(* Logix 5000 project; controller reports 1756-L63 rev 20.15; software revision 20.04; part 13 of 52 *)

        [466].log_data[0].valid := 1, [466].log_data[1].valid := 1, [466].log_data[2].valid := 1, [466].log_data[3].valid := 1, [466].log_data[4].valid := 1, [466].log_data[5].valid := 1, [466].log_data[6].valid := 1, [466].log_data[7].valid := 1, [466].log_data[8].valid := 1, [466].log_data[9].valid := 1, [466].log_data[10].valid := 1, [466].log_data[11].valid := 1, [466].log_data[12].valid := 1, [466].log_data[13].valid := 1, [466].log_data[14].valid := 1, [466].log_data[15].valid := 1, [466].log_data[16].valid := 1, [466].log_data[17].valid := 1, [466].log_data[18].valid := 1, [466].log_data[19].valid := 1, [466].time.Year := 2023, [466].time.Month := 1, [466].time.Day := 19, [466].time.Hour := 15, [466].time.Minute := 14, [466].time.Second := 59, [467].log_data[0].min := 1.0, [467].log_data[0].max := 1.0, [467].log_data[0].total := 300.0, [467].log_data[0].time := 300.0, [467].log_data[0].minminute := 15, [467].log_data[0].maxminute := 15, [467].log_data[0].valid := 1, [467].log_data[1].valid := 1, [467].log_data[2].valid := 1, [467].log_data[3].valid := 1, [467].log_data[4].valid := 1, [467].log_data[5].valid := 1, [467].log_data[6].valid := 1, [467].log_data[7].valid := 1, [467].log_data[8].valid := 1, [467].log_data[9].valid := 1, [467].log_data[10].valid := 1, [467].log_data[11].valid := 1, [467].log_data[12].valid := 1, [467].log_data[13].valid := 1, [467].log_data[14].valid := 1, [467].log_data[15].valid := 1, [467].log_data[16].valid := 1, [467].log_data[17].valid := 1, [467].log_data[18].valid := 1, [467].log_data[19].valid := 1, [467].time.Year := 2023, [467].time.Month := 1, [467].time.Day := 19, [467].time.Hour := 15, [467].time.Minute := 19, [467].time.Second := 59, [468].log_data[0].min := 1.0, [468].log_data[0].max := 1.0,
        [468].log_data[0].total := 300.0, [468].log_data[0].time := 300.0, [468].log_data[0].minminute := 20, [468].log_data[0].maxminute := 20, [468].log_data[0].valid := 1, [468].log_data[1].valid := 1, [468].log_data[2].valid := 1, [468].log_data[3].valid := 1, [468].log_data[4].valid := 1, [468].log_data[5].valid := 1, [468].log_data[6].valid := 1, [468].log_data[7].valid := 1, [468].log_data[8].valid := 1, [468].log_data[9].valid := 1, [468].log_data[10].valid := 1, [468].log_data[11].valid := 1, [468].log_data[12].valid := 1, [468].log_data[13].valid := 1, [468].log_data[14].valid := 1, [468].log_data[15].valid := 1, [468].log_data[16].valid := 1, [468].log_data[17].valid := 1, [468].log_data[18].valid := 1, [468].log_data[19].valid := 1, [468].time.Year := 2023, [468].time.Month := 1, [468].time.Day := 19, [468].time.Hour := 15, [468].time.Minute := 24, [468].time.Second := 59, [469].log_data[0].min := 1.0, [469].log_data[0].max := 1.0, [469].log_data[0].total := 44.5, [469].log_data[0].time := 44.5, [469].log_data[0].minminute := 25, [469].log_data[0].maxminute := 25, [469].log_data[0].valid := 1, [469].log_data[1].valid := 1, [469].log_data[2].valid := 1, [469].log_data[3].valid := 1, [469].log_data[4].valid := 1, [469].log_data[5].valid := 1, [469].log_data[6].valid := 1, [469].log_data[7].valid := 1, [469].log_data[8].valid := 1, [469].log_data[9].valid := 1, [469].log_data[10].valid := 1, [469].log_data[11].valid := 1, [469].log_data[12].valid := 1, [469].log_data[13].valid := 1, [469].log_data[14].valid := 1, [469].log_data[15].valid := 1, [469].log_data[16].valid := 1, [469].log_data[17].valid := 1, [469].log_data[18].valid := 1, [469].log_data[19].valid := 1, [470].log_data[0].min := 1.0, [470].log_data[0].max := 1.0, [470].log_data[0].total := 300.0, [470].log_data[0].time := 300.0,
        [470].log_data[0].minminute := 30, [470].log_data[0].maxminute := 30, [470].log_data[0].valid := 1, [470].log_data[1].valid := 1, [470].log_data[2].valid := 1, [470].log_data[3].valid := 1, [470].log_data[4].valid := 1, [470].log_data[5].valid := 1, [470].log_data[6].valid := 1, [470].log_data[7].valid := 1, [470].log_data[8].valid := 1, [470].log_data[9].valid := 1, [470].log_data[10].valid := 1, [470].log_data[11].valid := 1, [470].log_data[12].valid := 1, [470].log_data[13].valid := 1, [470].log_data[14].valid := 1, [470].log_data[15].valid := 1, [470].log_data[16].valid := 1, [470].log_data[17].valid := 1, [470].log_data[18].valid := 1, [470].log_data[19].valid := 1, [470].time.Year := 2023, [470].time.Month := 1, [470].time.Day := 11, [470].time.Hour := 7, [470].time.Minute := 34, [470].time.Second := 59, [471].log_data[0].min := 1.0, [471].log_data[0].max := 1.0, [471].log_data[0].total := 300.0, [471].log_data[0].time := 300.0, [471].log_data[0].minminute := 35, [471].log_data[0].maxminute := 35, [471].log_data[0].valid := 1, [471].log_data[1].valid := 1, [471].log_data[2].valid := 1, [471].log_data[3].valid := 1, [471].log_data[4].valid := 1, [471].log_data[5].valid := 1, [471].log_data[6].valid := 1, [471].log_data[7].valid := 1, [471].log_data[8].valid := 1, [471].log_data[9].valid := 1, [471].log_data[10].valid := 1, [471].log_data[11].valid := 1, [471].log_data[12].valid := 1, [471].log_data[13].valid := 1, [471].log_data[14].valid := 1, [471].log_data[15].valid := 1, [471].log_data[16].valid := 1, [471].log_data[17].valid := 1, [471].log_data[18].valid := 1, [471].log_data[19].valid := 1, [471].time.Year := 2023, [471].time.Month := 1, [471].time.Day := 11, [471].time.Hour := 7, [471].time.Minute := 39, [471].time.Second := 59,
        [472].log_data[0].min := 1.0, [472].log_data[0].max := 1.0, [472].log_data[0].total := 300.0, [472].log_data[0].time := 300.0, [472].log_data[0].minminute := 40, [472].log_data[0].maxminute := 40, [472].log_data[0].valid := 1, [472].log_data[1].valid := 1, [472].log_data[2].valid := 1, [472].log_data[3].valid := 1, [472].log_data[4].valid := 1, [472].log_data[5].valid := 1, [472].log_data[6].valid := 1, [472].log_data[7].valid := 1, [472].log_data[8].valid := 1, [472].log_data[9].valid := 1, [472].log_data[10].valid := 1, [472].log_data[11].valid := 1, [472].log_data[12].valid := 1, [472].log_data[13].valid := 1, [472].log_data[14].valid := 1, [472].log_data[15].valid := 1, [472].log_data[16].valid := 1, [472].log_data[17].valid := 1, [472].log_data[18].valid := 1, [472].log_data[19].valid := 1, [472].time.Year := 2023, [472].time.Month := 1, [472].time.Day := 11, [472].time.Hour := 7, [472].time.Minute := 44, [472].time.Second := 59, [473].log_data[0].min := 1.0, [473].log_data[0].max := 1.0, [473].log_data[0].total := 300.0, [473].log_data[0].time := 300.0, [473].log_data[0].minminute := 45, [473].log_data[0].maxminute := 45, [473].log_data[0].valid := 1, [473].log_data[1].valid := 1, [473].log_data[2].valid := 1, [473].log_data[3].valid := 1, [473].log_data[4].valid := 1, [473].log_data[5].valid := 1, [473].log_data[6].valid := 1, [473].log_data[7].valid := 1, [473].log_data[8].valid := 1, [473].log_data[9].valid := 1, [473].log_data[10].valid := 1, [473].log_data[11].valid := 1, [473].log_data[12].valid := 1, [473].log_data[13].valid := 1, [473].log_data[14].valid := 1, [473].log_data[15].valid := 1, [473].log_data[16].valid := 1, [473].log_data[17].valid := 1, [473].log_data[18].valid := 1, [473].log_data[19].valid := 1, [473].time.Year := 2023, [473].time.Month := 1,
        [473].time.Day := 11, [473].time.Hour := 7, [473].time.Minute := 49, [473].time.Second := 59, [474].log_data[0].min := 1.0, [474].log_data[0].max := 1.0, [474].log_data[0].total := 300.0, [474].log_data[0].time := 300.0, [474].log_data[0].minminute := 50, [474].log_data[0].maxminute := 50, [474].log_data[0].valid := 1, [474].log_data[1].valid := 1, [474].log_data[2].valid := 1, [474].log_data[3].valid := 1, [474].log_data[4].valid := 1, [474].log_data[5].valid := 1, [474].log_data[6].valid := 1, [474].log_data[7].valid := 1, [474].log_data[8].valid := 1, [474].log_data[9].valid := 1, [474].log_data[10].valid := 1, [474].log_data[11].valid := 1, [474].log_data[12].valid := 1, [474].log_data[13].valid := 1, [474].log_data[14].valid := 1, [474].log_data[15].valid := 1, [474].log_data[16].valid := 1, [474].log_data[17].valid := 1, [474].log_data[18].valid := 1, [474].log_data[19].valid := 1, [474].time.Year := 2023, [474].time.Month := 1, [474].time.Day := 11, [474].time.Hour := 7, [474].time.Minute := 54, [474].time.Second := 59, [475].log_data[0].min := 1.0, [475].log_data[0].max := 1.0, [475].log_data[0].total := 300.0, [475].log_data[0].time := 300.0, [475].log_data[0].minminute := 55, [475].log_data[0].maxminute := 55, [475].log_data[0].valid := 1, [475].log_data[1].valid := 1, [475].log_data[2].valid := 1, [475].log_data[3].valid := 1, [475].log_data[4].valid := 1, [475].log_data[5].valid := 1, [475].log_data[6].valid := 1, [475].log_data[7].valid := 1, [475].log_data[8].valid := 1, [475].log_data[9].valid := 1, [475].log_data[10].valid := 1, [475].log_data[11].valid := 1, [475].log_data[12].valid := 1, [475].log_data[13].valid := 1, [475].log_data[14].valid := 1, [475].log_data[15].valid := 1, [475].log_data[16].valid := 1, [475].log_data[17].valid := 1,
        [475].log_data[18].valid := 1, [475].log_data[19].valid := 1, [475].time.Year := 2023, [475].time.Month := 1, [475].time.Day := 11, [475].time.Hour := 7, [475].time.Minute := 59, [475].time.Second := 59, [476].log_data[0].min := 1.0, [476].log_data[0].max := 1.0, [476].log_data[0].total := 300.0, [476].log_data[0].time := 300.0, [476].log_data[0].valid := 1, [476].log_data[1].valid := 1, [476].log_data[2].valid := 1, [476].log_data[3].valid := 1, [476].log_data[4].valid := 1, [476].log_data[5].valid := 1, [476].log_data[6].valid := 1, [476].log_data[7].valid := 1, [476].log_data[8].valid := 1, [476].log_data[9].valid := 1, [476].log_data[10].valid := 1, [476].log_data[11].valid := 1, [476].log_data[12].valid := 1, [476].log_data[13].valid := 1, [476].log_data[14].valid := 1, [476].log_data[15].valid := 1, [476].log_data[16].valid := 1, [476].log_data[17].valid := 1, [476].log_data[18].valid := 1, [476].log_data[19].valid := 1, [476].time.Year := 2023, [476].time.Month := 1, [476].time.Day := 11, [476].time.Hour := 8, [476].time.Minute := 4, [476].time.Second := 59, [477].log_data[0].min := 1.0, [477].log_data[0].max := 1.0, [477].log_data[0].total := 300.0, [477].log_data[0].time := 300.0, [477].log_data[0].minminute := 5, [477].log_data[0].maxminute := 5, [477].log_data[0].valid := 1, [477].log_data[1].valid := 1, [477].log_data[2].valid := 1, [477].log_data[3].valid := 1, [477].log_data[4].valid := 1, [477].log_data[5].valid := 1, [477].log_data[6].valid := 1, [477].log_data[7].valid := 1, [477].log_data[8].valid := 1, [477].log_data[9].valid := 1, [477].log_data[10].valid := 1, [477].log_data[11].valid := 1, [477].log_data[12].valid := 1, [477].log_data[13].valid := 1, [477].log_data[14].valid := 1, [477].log_data[15].valid := 1,
        [477].log_data[16].valid := 1, [477].log_data[17].valid := 1, [477].log_data[18].valid := 1, [477].log_data[19].valid := 1, [477].time.Year := 2023, [477].time.Month := 1, [477].time.Day := 11, [477].time.Hour := 8, [477].time.Minute := 9, [477].time.Second := 59, [478].log_data[0].min := 1.0, [478].log_data[0].max := 1.0, [478].log_data[0].total := 300.0, [478].log_data[0].time := 300.0, [478].log_data[0].minminute := 10, [478].log_data[0].maxminute := 10, [478].log_data[0].valid := 1, [478].log_data[1].valid := 1, [478].log_data[2].valid := 1, [478].log_data[3].valid := 1, [478].log_data[4].valid := 1, [478].log_data[5].valid := 1, [478].log_data[6].valid := 1, [478].log_data[7].valid := 1, [478].log_data[8].valid := 1, [478].log_data[9].valid := 1, [478].log_data[10].valid := 1, [478].log_data[11].valid := 1, [478].log_data[12].valid := 1, [478].log_data[13].valid := 1, [478].log_data[14].valid := 1, [478].log_data[15].valid := 1, [478].log_data[16].valid := 1, [478].log_data[17].valid := 1, [478].log_data[18].valid := 1, [478].log_data[19].valid := 1, [478].time.Year := 2023, [478].time.Month := 1, [478].time.Day := 11, [478].time.Hour := 8, [478].time.Minute := 14, [478].time.Second := 59, [479].log_data[0].min := 1.0, [479].log_data[0].max := 1.0, [479].log_data[0].total := 300.0, [479].log_data[0].time := 300.0, [479].log_data[0].minminute := 15, [479].log_data[0].maxminute := 15, [479].log_data[0].valid := 1, [479].log_data[1].valid := 1, [479].log_data[2].valid := 1, [479].log_data[3].valid := 1, [479].log_data[4].valid := 1, [479].log_data[5].valid := 1, [479].log_data[6].valid := 1, [479].log_data[7].valid := 1, [479].log_data[8].valid := 1, [479].log_data[9].valid := 1, [479].log_data[10].valid := 1, [479].log_data[11].valid := 1,
        [479].log_data[12].valid := 1, [479].log_data[13].valid := 1, [479].log_data[14].valid := 1, [479].log_data[15].valid := 1, [479].log_data[16].valid := 1, [479].log_data[17].valid := 1, [479].log_data[18].valid := 1, [479].log_data[19].valid := 1, [479].time.Year := 2023, [479].time.Month := 1, [479].time.Day := 11, [479].time.Hour := 8, [479].time.Minute := 19, [479].time.Second := 59, [480].log_data[0].min := 1.0, [480].log_data[0].max := 1.0, [480].log_data[0].total := 300.0, [480].log_data[0].time := 300.0, [480].log_data[0].minminute := 20, [480].log_data[0].maxminute := 20, [480].log_data[0].valid := 1, [480].log_data[1].valid := 1, [480].log_data[2].valid := 1, [480].log_data[3].valid := 1, [480].log_data[4].valid := 1, [480].log_data[5].valid := 1, [480].log_data[6].valid := 1, [480].log_data[7].valid := 1, [480].log_data[8].valid := 1, [480].log_data[9].valid := 1, [480].log_data[10].valid := 1, [480].log_data[11].valid := 1, [480].log_data[12].valid := 1, [480].log_data[13].valid := 1, [480].log_data[14].valid := 1, [480].log_data[15].valid := 1, [480].log_data[16].valid := 1, [480].log_data[17].valid := 1, [480].log_data[18].valid := 1, [480].log_data[19].valid := 1, [480].time.Year := 2023, [480].time.Month := 1, [480].time.Day := 11, [480].time.Hour := 8, [480].time.Minute := 24, [480].time.Second := 59, [481].log_data[0].min := 1.0, [481].log_data[0].max := 1.0, [481].log_data[0].total := 300.0, [481].log_data[0].time := 300.0, [481].log_data[0].minminute := 25, [481].log_data[0].maxminute := 25, [481].log_data[0].valid := 1, [481].log_data[1].valid := 1, [481].log_data[2].valid := 1, [481].log_data[3].valid := 1, [481].log_data[4].valid := 1, [481].log_data[5].valid := 1, [481].log_data[6].valid := 1, [481].log_data[7].valid := 1,
        [481].log_data[8].valid := 1, [481].log_data[9].valid := 1, [481].log_data[10].valid := 1, [481].log_data[11].valid := 1, [481].log_data[12].valid := 1, [481].log_data[13].valid := 1, [481].log_data[14].valid := 1, [481].log_data[15].valid := 1, [481].log_data[16].valid := 1, [481].log_data[17].valid := 1, [481].log_data[18].valid := 1, [481].log_data[19].valid := 1, [481].time.Year := 2023, [481].time.Month := 1, [481].time.Day := 11, [481].time.Hour := 8, [481].time.Minute := 29, [481].time.Second := 59, [482].log_data[0].min := 1.0, [482].log_data[0].max := 1.0, [482].log_data[0].total := 300.0, [482].log_data[0].time := 300.0, [482].log_data[0].minminute := 30, [482].log_data[0].maxminute := 30, [482].log_data[0].valid := 1, [482].log_data[1].valid := 1, [482].log_data[2].valid := 1, [482].log_data[3].valid := 1, [482].log_data[4].valid := 1, [482].log_data[5].valid := 1, [482].log_data[6].valid := 1, [482].log_data[7].valid := 1, [482].log_data[8].valid := 1, [482].log_data[9].valid := 1, [482].log_data[10].valid := 1, [482].log_data[11].valid := 1, [482].log_data[12].valid := 1, [482].log_data[13].valid := 1, [482].log_data[14].valid := 1, [482].log_data[15].valid := 1, [482].log_data[16].valid := 1, [482].log_data[17].valid := 1, [482].log_data[18].valid := 1, [482].log_data[19].valid := 1, [482].time.Year := 2023, [482].time.Month := 1, [482].time.Day := 11, [482].time.Hour := 8, [482].time.Minute := 34, [482].time.Second := 59, [483].log_data[0].min := 1.0, [483].log_data[0].max := 1.0, [483].log_data[0].total := 300.0, [483].log_data[0].time := 300.0, [483].log_data[0].minminute := 35, [483].log_data[0].maxminute := 35, [483].log_data[0].valid := 1, [483].log_data[1].valid := 1, [483].log_data[2].valid := 1, [483].log_data[3].valid := 1,
        [483].log_data[4].valid := 1, [483].log_data[5].valid := 1, [483].log_data[6].valid := 1, [483].log_data[7].valid := 1, [483].log_data[8].valid := 1, [483].log_data[9].valid := 1, [483].log_data[10].valid := 1, [483].log_data[11].valid := 1, [483].log_data[12].valid := 1, [483].log_data[13].valid := 1, [483].log_data[14].valid := 1, [483].log_data[15].valid := 1, [483].log_data[16].valid := 1, [483].log_data[17].valid := 1, [483].log_data[18].valid := 1, [483].log_data[19].valid := 1, [483].time.Year := 2023, [483].time.Month := 1, [483].time.Day := 11, [483].time.Hour := 8, [483].time.Minute := 39, [483].time.Second := 59, [484].log_data[0].min := 1.0, [484].log_data[0].max := 1.0, [484].log_data[0].total := 300.0, [484].log_data[0].time := 300.0, [484].log_data[0].minminute := 40, [484].log_data[0].maxminute := 40, [484].log_data[0].valid := 1, [484].log_data[1].valid := 1, [484].log_data[2].valid := 1, [484].log_data[3].valid := 1, [484].log_data[4].valid := 1, [484].log_data[5].valid := 1, [484].log_data[6].valid := 1, [484].log_data[7].valid := 1, [484].log_data[8].valid := 1, [484].log_data[9].valid := 1, [484].log_data[10].valid := 1, [484].log_data[11].valid := 1, [484].log_data[12].valid := 1, [484].log_data[13].valid := 1, [484].log_data[14].valid := 1, [484].log_data[15].valid := 1, [484].log_data[16].valid := 1, [484].log_data[17].valid := 1, [484].log_data[18].valid := 1, [484].log_data[19].valid := 1, [484].time.Year := 2023, [484].time.Month := 1, [484].time.Day := 11, [484].time.Hour := 8, [484].time.Minute := 44, [484].time.Second := 59, [485].log_data[0].min := 1.0, [485].log_data[0].max := 1.0, [485].log_data[0].total := 300.0, [485].log_data[0].time := 300.0, [485].log_data[0].minminute := 45, [485].log_data[0].maxminute := 45,
        [485].log_data[0].valid := 1, [485].log_data[1].valid := 1, [485].log_data[2].valid := 1, [485].log_data[3].valid := 1, [485].log_data[4].valid := 1, [485].log_data[5].valid := 1, [485].log_data[6].valid := 1, [485].log_data[7].valid := 1, [485].log_data[8].valid := 1, [485].log_data[9].valid := 1, [485].log_data[10].valid := 1, [485].log_data[11].valid := 1, [485].log_data[12].valid := 1, [485].log_data[13].valid := 1, [485].log_data[14].valid := 1, [485].log_data[15].valid := 1, [485].log_data[16].valid := 1, [485].log_data[17].valid := 1, [485].log_data[18].valid := 1, [485].log_data[19].valid := 1, [485].time.Year := 2023, [485].time.Month := 1, [485].time.Day := 11, [485].time.Hour := 8, [485].time.Minute := 49, [485].time.Second := 59, [486].log_data[0].min := 1.0, [486].log_data[0].max := 1.0, [486].log_data[0].total := 300.0, [486].log_data[0].time := 300.0, [486].log_data[0].minminute := 50, [486].log_data[0].maxminute := 50, [486].log_data[0].valid := 1, [486].log_data[1].valid := 1, [486].log_data[2].valid := 1, [486].log_data[3].valid := 1, [486].log_data[4].valid := 1, [486].log_data[5].valid := 1, [486].log_data[6].valid := 1, [486].log_data[7].valid := 1, [486].log_data[8].valid := 1, [486].log_data[9].valid := 1, [486].log_data[10].valid := 1, [486].log_data[11].valid := 1, [486].log_data[12].valid := 1, [486].log_data[13].valid := 1, [486].log_data[14].valid := 1, [486].log_data[15].valid := 1, [486].log_data[16].valid := 1, [486].log_data[17].valid := 1, [486].log_data[18].valid := 1, [486].log_data[19].valid := 1, [486].time.Year := 2023, [486].time.Month := 1, [486].time.Day := 11, [486].time.Hour := 8, [486].time.Minute := 54, [486].time.Second := 59, [487].log_data[0].min := 1.0, [487].log_data[0].max := 1.0,
        [487].log_data[0].total := 300.0, [487].log_data[0].time := 300.0, [487].log_data[0].minminute := 55, [487].log_data[0].maxminute := 55, [487].log_data[0].valid := 1, [487].log_data[1].valid := 1, [487].log_data[2].valid := 1, [487].log_data[3].valid := 1, [487].log_data[4].valid := 1, [487].log_data[5].valid := 1, [487].log_data[6].valid := 1, [487].log_data[7].valid := 1, [487].log_data[8].valid := 1, [487].log_data[9].valid := 1, [487].log_data[10].valid := 1, [487].log_data[11].valid := 1, [487].log_data[12].valid := 1, [487].log_data[13].valid := 1, [487].log_data[14].valid := 1, [487].log_data[15].valid := 1, [487].log_data[16].valid := 1, [487].log_data[17].valid := 1, [487].log_data[18].valid := 1, [487].log_data[19].valid := 1, [487].time.Year := 2023, [487].time.Month := 1, [487].time.Day := 11, [487].time.Hour := 8, [487].time.Minute := 59, [487].time.Second := 59, [488].log_data[0].min := 1.0, [488].log_data[0].max := 1.0, [488].log_data[0].total := 300.0, [488].log_data[0].time := 300.0, [488].log_data[0].valid := 1, [488].log_data[1].valid := 1, [488].log_data[2].valid := 1, [488].log_data[3].valid := 1, [488].log_data[4].valid := 1, [488].log_data[5].valid := 1, [488].log_data[6].valid := 1, [488].log_data[7].valid := 1, [488].log_data[8].valid := 1, [488].log_data[9].valid := 1, [488].log_data[10].valid := 1, [488].log_data[11].valid := 1, [488].log_data[12].valid := 1, [488].log_data[13].valid := 1, [488].log_data[14].valid := 1, [488].log_data[15].valid := 1, [488].log_data[16].valid := 1, [488].log_data[17].valid := 1, [488].log_data[18].valid := 1, [488].log_data[19].valid := 1, [488].time.Year := 2023, [488].time.Month := 1, [488].time.Day := 11, [488].time.Hour := 9, [488].time.Minute := 4, [488].time.Second := 59,
        [489].log_data[0].min := 1.0, [489].log_data[0].max := 1.0, [489].log_data[0].total := 300.0, [489].log_data[0].time := 300.0, [489].log_data[0].minminute := 5, [489].log_data[0].maxminute := 5, [489].log_data[0].valid := 1, [489].log_data[1].valid := 1, [489].log_data[2].valid := 1, [489].log_data[3].valid := 1, [489].log_data[4].valid := 1, [489].log_data[5].valid := 1, [489].log_data[6].valid := 1, [489].log_data[7].valid := 1, [489].log_data[8].valid := 1, [489].log_data[9].valid := 1, [489].log_data[10].valid := 1, [489].log_data[11].valid := 1, [489].log_data[12].valid := 1, [489].log_data[13].valid := 1, [489].log_data[14].valid := 1, [489].log_data[15].valid := 1, [489].log_data[16].valid := 1, [489].log_data[17].valid := 1, [489].log_data[18].valid := 1, [489].log_data[19].valid := 1, [489].time.Year := 2023, [489].time.Month := 1, [489].time.Day := 11, [489].time.Hour := 9, [489].time.Minute := 9, [489].time.Second := 59, [490].log_data[0].min := 1.0, [490].log_data[0].max := 1.0, [490].log_data[0].total := 300.0, [490].log_data[0].time := 300.0, [490].log_data[0].minminute := 10, [490].log_data[0].maxminute := 10, [490].log_data[0].valid := 1, [490].log_data[1].valid := 1, [490].log_data[2].valid := 1, [490].log_data[3].valid := 1, [490].log_data[4].valid := 1, [490].log_data[5].valid := 1, [490].log_data[6].valid := 1, [490].log_data[7].valid := 1, [490].log_data[8].valid := 1, [490].log_data[9].valid := 1, [490].log_data[10].valid := 1, [490].log_data[11].valid := 1, [490].log_data[12].valid := 1, [490].log_data[13].valid := 1, [490].log_data[14].valid := 1, [490].log_data[15].valid := 1, [490].log_data[16].valid := 1, [490].log_data[17].valid := 1, [490].log_data[18].valid := 1, [490].log_data[19].valid := 1, [490].time.Year := 2023, [490].time.Month := 1,
        [490].time.Day := 11, [490].time.Hour := 9, [490].time.Minute := 14, [490].time.Second := 59, [491].log_data[0].min := 1.0, [491].log_data[0].max := 1.0, [491].log_data[0].total := 300.0, [491].log_data[0].time := 300.0, [491].log_data[0].minminute := 15, [491].log_data[0].maxminute := 15, [491].log_data[0].valid := 1, [491].log_data[1].valid := 1, [491].log_data[2].valid := 1, [491].log_data[3].valid := 1, [491].log_data[4].valid := 1, [491].log_data[5].valid := 1, [491].log_data[6].valid := 1, [491].log_data[7].valid := 1, [491].log_data[8].valid := 1, [491].log_data[9].valid := 1, [491].log_data[10].valid := 1, [491].log_data[11].valid := 1, [491].log_data[12].valid := 1, [491].log_data[13].valid := 1, [491].log_data[14].valid := 1, [491].log_data[15].valid := 1, [491].log_data[16].valid := 1, [491].log_data[17].valid := 1, [491].log_data[18].valid := 1, [491].log_data[19].valid := 1, [491].time.Year := 2023, [491].time.Month := 1, [491].time.Day := 11, [491].time.Hour := 9, [491].time.Minute := 19, [491].time.Second := 59, [492].log_data[0].min := 1.0, [492].log_data[0].max := 1.0, [492].log_data[0].total := 300.0, [492].log_data[0].time := 300.0, [492].log_data[0].minminute := 20, [492].log_data[0].maxminute := 20, [492].log_data[0].valid := 1, [492].log_data[1].valid := 1, [492].log_data[2].valid := 1, [492].log_data[3].valid := 1, [492].log_data[4].valid := 1, [492].log_data[5].valid := 1, [492].log_data[6].valid := 1, [492].log_data[7].valid := 1, [492].log_data[8].valid := 1, [492].log_data[9].valid := 1, [492].log_data[10].valid := 1, [492].log_data[11].valid := 1, [492].log_data[12].valid := 1, [492].log_data[13].valid := 1, [492].log_data[14].valid := 1, [492].log_data[15].valid := 1, [492].log_data[16].valid := 1, [492].log_data[17].valid := 1,
        [492].log_data[18].valid := 1, [492].log_data[19].valid := 1, [492].time.Year := 2023, [492].time.Month := 1, [492].time.Day := 11, [492].time.Hour := 9, [492].time.Minute := 24, [492].time.Second := 59, [493].log_data[0].min := 1.0, [493].log_data[0].max := 1.0, [493].log_data[0].total := 300.0, [493].log_data[0].time := 300.0, [493].log_data[0].minminute := 25, [493].log_data[0].maxminute := 25, [493].log_data[0].valid := 1, [493].log_data[1].valid := 1, [493].log_data[2].valid := 1, [493].log_data[3].valid := 1, [493].log_data[4].valid := 1, [493].log_data[5].valid := 1, [493].log_data[6].valid := 1, [493].log_data[7].valid := 1, [493].log_data[8].valid := 1, [493].log_data[9].valid := 1, [493].log_data[10].valid := 1, [493].log_data[11].valid := 1, [493].log_data[12].valid := 1, [493].log_data[13].valid := 1, [493].log_data[14].valid := 1, [493].log_data[15].valid := 1, [493].log_data[16].valid := 1, [493].log_data[17].valid := 1, [493].log_data[18].valid := 1, [493].log_data[19].valid := 1, [493].time.Year := 2023, [493].time.Month := 1, [493].time.Day := 11, [493].time.Hour := 9, [493].time.Minute := 29, [493].time.Second := 59, [494].log_data[0].min := 1.0, [494].log_data[0].max := 1.0, [494].log_data[0].total := 300.0, [494].log_data[0].time := 300.0, [494].log_data[0].minminute := 30, [494].log_data[0].maxminute := 30, [494].log_data[0].valid := 1, [494].log_data[1].valid := 1, [494].log_data[2].valid := 1, [494].log_data[3].valid := 1, [494].log_data[4].valid := 1, [494].log_data[5].valid := 1, [494].log_data[6].valid := 1, [494].log_data[7].valid := 1, [494].log_data[8].valid := 1, [494].log_data[9].valid := 1, [494].log_data[10].valid := 1, [494].log_data[11].valid := 1, [494].log_data[12].valid := 1, [494].log_data[13].valid := 1,
        [494].log_data[14].valid := 1, [494].log_data[15].valid := 1, [494].log_data[16].valid := 1, [494].log_data[17].valid := 1, [494].log_data[18].valid := 1, [494].log_data[19].valid := 1, [494].time.Year := 2023, [494].time.Month := 1, [494].time.Day := 11, [494].time.Hour := 9, [494].time.Minute := 34, [494].time.Second := 59, [495].log_data[0].min := 1.0, [495].log_data[0].max := 1.0, [495].log_data[0].total := 300.0, [495].log_data[0].time := 300.0, [495].log_data[0].minminute := 35, [495].log_data[0].maxminute := 35, [495].log_data[0].valid := 1, [495].log_data[1].valid := 1, [495].log_data[2].valid := 1, [495].log_data[3].valid := 1, [495].log_data[4].valid := 1, [495].log_data[5].valid := 1, [495].log_data[6].valid := 1, [495].log_data[7].valid := 1, [495].log_data[8].valid := 1, [495].log_data[9].valid := 1, [495].log_data[10].valid := 1, [495].log_data[11].valid := 1, [495].log_data[12].valid := 1, [495].log_data[13].valid := 1, [495].log_data[14].valid := 1, [495].log_data[15].valid := 1, [495].log_data[16].valid := 1, [495].log_data[17].valid := 1, [495].log_data[18].valid := 1, [495].log_data[19].valid := 1, [495].time.Year := 2023, [495].time.Month := 1, [495].time.Day := 11, [495].time.Hour := 9, [495].time.Minute := 39, [495].time.Second := 59, [496].log_data[0].min := 1.0, [496].log_data[0].max := 1.0, [496].log_data[0].total := 300.0, [496].log_data[0].time := 300.0, [496].log_data[0].minminute := 40, [496].log_data[0].maxminute := 40, [496].log_data[0].valid := 1, [496].log_data[1].valid := 1, [496].log_data[2].valid := 1, [496].log_data[3].valid := 1, [496].log_data[4].valid := 1, [496].log_data[5].valid := 1, [496].log_data[6].valid := 1, [496].log_data[7].valid := 1, [496].log_data[8].valid := 1, [496].log_data[9].valid := 1,
        [496].log_data[10].valid := 1, [496].log_data[11].valid := 1, [496].log_data[12].valid := 1, [496].log_data[13].valid := 1, [496].log_data[14].valid := 1, [496].log_data[15].valid := 1, [496].log_data[16].valid := 1, [496].log_data[17].valid := 1, [496].log_data[18].valid := 1, [496].log_data[19].valid := 1, [496].time.Year := 2023, [496].time.Month := 1, [496].time.Day := 11, [496].time.Hour := 9, [496].time.Minute := 44, [496].time.Second := 59, [497].log_data[0].min := 1.0, [497].log_data[0].max := 1.0, [497].log_data[0].total := 300.0, [497].log_data[0].time := 300.0, [497].log_data[0].minminute := 45, [497].log_data[0].maxminute := 45, [497].log_data[0].valid := 1, [497].log_data[1].valid := 1, [497].log_data[2].valid := 1, [497].log_data[3].valid := 1, [497].log_data[4].valid := 1, [497].log_data[5].valid := 1, [497].log_data[6].valid := 1, [497].log_data[7].valid := 1, [497].log_data[8].valid := 1, [497].log_data[9].valid := 1, [497].log_data[10].valid := 1, [497].log_data[11].valid := 1, [497].log_data[12].valid := 1, [497].log_data[13].valid := 1, [497].log_data[14].valid := 1, [497].log_data[15].valid := 1, [497].log_data[16].valid := 1, [497].log_data[17].valid := 1, [497].log_data[18].valid := 1, [497].log_data[19].valid := 1, [497].time.Year := 2023, [497].time.Month := 1, [497].time.Day := 11, [497].time.Hour := 9, [497].time.Minute := 49, [497].time.Second := 59, [498].log_data[0].min := 1.0, [498].log_data[0].max := 1.0, [498].log_data[0].total := 300.0, [498].log_data[0].time := 300.0, [498].log_data[0].minminute := 50, [498].log_data[0].maxminute := 50, [498].log_data[0].valid := 1, [498].log_data[1].valid := 1, [498].log_data[2].valid := 1, [498].log_data[3].valid := 1, [498].log_data[4].valid := 1, [498].log_data[5].valid := 1,
        [498].log_data[6].valid := 1, [498].log_data[7].valid := 1, [498].log_data[8].valid := 1, [498].log_data[9].valid := 1, [498].log_data[10].valid := 1, [498].log_data[11].valid := 1, [498].log_data[12].valid := 1, [498].log_data[13].valid := 1, [498].log_data[14].valid := 1, [498].log_data[15].valid := 1, [498].log_data[16].valid := 1, [498].log_data[17].valid := 1, [498].log_data[18].valid := 1, [498].log_data[19].valid := 1, [498].time.Year := 2023, [498].time.Month := 1, [498].time.Day := 11, [498].time.Hour := 9, [498].time.Minute := 54, [498].time.Second := 59, [499].log_data[0].min := 1.0, [499].log_data[0].max := 1.0, [499].log_data[0].total := 300.0, [499].log_data[0].time := 300.0, [499].log_data[0].minminute := 55, [499].log_data[0].maxminute := 55, [499].log_data[0].valid := 1, [499].log_data[1].valid := 1, [499].log_data[2].valid := 1, [499].log_data[3].valid := 1, [499].log_data[4].valid := 1, [499].log_data[5].valid := 1, [499].log_data[6].valid := 1, [499].log_data[7].valid := 1, [499].log_data[8].valid := 1, [499].log_data[9].valid := 1, [499].log_data[10].valid := 1, [499].log_data[11].valid := 1, [499].log_data[12].valid := 1, [499].log_data[13].valid := 1, [499].log_data[14].valid := 1, [499].log_data[15].valid := 1, [499].log_data[16].valid := 1, [499].log_data[17].valid := 1, [499].log_data[18].valid := 1, [499].log_data[19].valid := 1, [499].time.Year := 2023, [499].time.Month := 1, [499].time.Day := 11, [499].time.Hour := 9, [499].time.Minute := 59, [499].time.Second := 59, [500].log_data[0].min := 1.0, [500].log_data[0].max := 1.0, [500].log_data[0].total := 300.0, [500].log_data[0].time := 300.0, [500].log_data[0].valid := 1, [500].log_data[1].valid := 1, [500].log_data[2].valid := 1, [500].log_data[3].valid := 1,
        [500].log_data[4].valid := 1, [500].log_data[5].valid := 1, [500].log_data[6].valid := 1, [500].log_data[7].valid := 1, [500].log_data[8].valid := 1, [500].log_data[9].valid := 1, [500].log_data[10].valid := 1, [500].log_data[11].valid := 1, [500].log_data[12].valid := 1, [500].log_data[13].valid := 1, [500].log_data[14].valid := 1, [500].log_data[15].valid := 1, [500].log_data[16].valid := 1, [500].log_data[17].valid := 1, [500].log_data[18].valid := 1, [500].log_data[19].valid := 1, [500].time.Year := 2023, [500].time.Month := 1, [500].time.Day := 11, [500].time.Hour := 10, [500].time.Minute := 4, [500].time.Second := 59, [501].log_data[0].min := 1.0, [501].log_data[0].max := 1.0, [501].log_data[0].total := 300.0, [501].log_data[0].time := 300.0, [501].log_data[0].minminute := 5, [501].log_data[0].maxminute := 5, [501].log_data[0].valid := 1, [501].log_data[1].valid := 1, [501].log_data[2].valid := 1, [501].log_data[3].valid := 1, [501].log_data[4].valid := 1, [501].log_data[5].valid := 1, [501].log_data[6].valid := 1, [501].log_data[7].valid := 1, [501].log_data[8].valid := 1, [501].log_data[9].valid := 1, [501].log_data[10].valid := 1, [501].log_data[11].valid := 1, [501].log_data[12].valid := 1, [501].log_data[13].valid := 1, [501].log_data[14].valid := 1, [501].log_data[15].valid := 1, [501].log_data[16].valid := 1, [501].log_data[17].valid := 1, [501].log_data[18].valid := 1, [501].log_data[19].valid := 1, [501].time.Year := 2023, [501].time.Month := 1, [501].time.Day := 11, [501].time.Hour := 10, [501].time.Minute := 9, [501].time.Second := 59, [502].log_data[0].min := 1.0, [502].log_data[0].max := 1.0, [502].log_data[0].total := 300.0, [502].log_data[0].time := 300.0, [502].log_data[0].minminute := 10, [502].log_data[0].maxminute := 10,
        [502].log_data[0].valid := 1, [502].log_data[1].valid := 1, [502].log_data[2].valid := 1, [502].log_data[3].valid := 1, [502].log_data[4].valid := 1, [502].log_data[5].valid := 1, [502].log_data[6].valid := 1, [502].log_data[7].valid := 1, [502].log_data[8].valid := 1, [502].log_data[9].valid := 1, [502].log_data[10].valid := 1, [502].log_data[11].valid := 1, [502].log_data[12].valid := 1, [502].log_data[13].valid := 1, [502].log_data[14].valid := 1, [502].log_data[15].valid := 1, [502].log_data[16].valid := 1, [502].log_data[17].valid := 1, [502].log_data[18].valid := 1, [502].log_data[19].valid := 1, [502].time.Year := 2023, [502].time.Month := 1, [502].time.Day := 11, [502].time.Hour := 10, [502].time.Minute := 14, [502].time.Second := 59, [503].log_data[0].min := 1.0, [503].log_data[0].max := 1.0, [503].log_data[0].total := 300.0, [503].log_data[0].time := 300.0, [503].log_data[0].minminute := 15, [503].log_data[0].maxminute := 15, [503].log_data[0].valid := 1, [503].log_data[1].valid := 1, [503].log_data[2].valid := 1, [503].log_data[3].valid := 1, [503].log_data[4].valid := 1, [503].log_data[5].valid := 1, [503].log_data[6].valid := 1, [503].log_data[7].valid := 1, [503].log_data[8].valid := 1, [503].log_data[9].valid := 1, [503].log_data[10].valid := 1, [503].log_data[11].valid := 1, [503].log_data[12].valid := 1, [503].log_data[13].valid := 1, [503].log_data[14].valid := 1, [503].log_data[15].valid := 1, [503].log_data[16].valid := 1, [503].log_data[17].valid := 1, [503].log_data[18].valid := 1, [503].log_data[19].valid := 1, [503].time.Year := 2023, [503].time.Month := 1, [503].time.Day := 11, [503].time.Hour := 10, [503].time.Minute := 19, [503].time.Second := 59, [504].log_data[0].min := 1.0, [504].log_data[0].max := 1.0,
        [504].log_data[0].total := 300.0, [504].log_data[0].time := 300.0, [504].log_data[0].minminute := 20, [504].log_data[0].maxminute := 20, [504].log_data[0].valid := 1, [504].log_data[1].valid := 1, [504].log_data[2].valid := 1, [504].log_data[3].valid := 1, [504].log_data[4].valid := 1, [504].log_data[5].valid := 1, [504].log_data[6].valid := 1, [504].log_data[7].valid := 1, [504].log_data[8].valid := 1, [504].log_data[9].valid := 1, [504].log_data[10].valid := 1, [504].log_data[11].valid := 1, [504].log_data[12].valid := 1, [504].log_data[13].valid := 1, [504].log_data[14].valid := 1, [504].log_data[15].valid := 1, [504].log_data[16].valid := 1, [504].log_data[17].valid := 1, [504].log_data[18].valid := 1, [504].log_data[19].valid := 1, [504].time.Year := 2023, [504].time.Month := 1, [504].time.Day := 11, [504].time.Hour := 10, [504].time.Minute := 24, [504].time.Second := 59, [505].log_data[0].min := 1.0, [505].log_data[0].max := 1.0, [505].log_data[0].total := 300.0, [505].log_data[0].time := 300.0, [505].log_data[0].minminute := 25, [505].log_data[0].maxminute := 25, [505].log_data[0].valid := 1, [505].log_data[1].valid := 1, [505].log_data[2].valid := 1, [505].log_data[3].valid := 1, [505].log_data[4].valid := 1, [505].log_data[5].valid := 1, [505].log_data[6].valid := 1, [505].log_data[7].valid := 1, [505].log_data[8].valid := 1, [505].log_data[9].valid := 1, [505].log_data[10].valid := 1, [505].log_data[11].valid := 1, [505].log_data[12].valid := 1, [505].log_data[13].valid := 1, [505].log_data[14].valid := 1, [505].log_data[15].valid := 1, [505].log_data[16].valid := 1, [505].log_data[17].valid := 1, [505].log_data[18].valid := 1, [505].log_data[19].valid := 1, [505].time.Year := 2023, [505].time.Month := 1, [505].time.Day := 11, [505].time.Hour := 10,
        [505].time.Minute := 29, [505].time.Second := 59, [506].log_data[0].min := 1.0, [506].log_data[0].max := 1.0, [506].log_data[0].total := 300.0, [506].log_data[0].time := 300.0, [506].log_data[0].minminute := 30, [506].log_data[0].maxminute := 30, [506].log_data[0].valid := 1, [506].log_data[1].valid := 1, [506].log_data[2].valid := 1, [506].log_data[3].valid := 1, [506].log_data[4].valid := 1, [506].log_data[5].valid := 1, [506].log_data[6].valid := 1, [506].log_data[7].valid := 1, [506].log_data[8].valid := 1, [506].log_data[9].valid := 1, [506].log_data[10].valid := 1, [506].log_data[11].valid := 1, [506].log_data[12].valid := 1, [506].log_data[13].valid := 1, [506].log_data[14].valid := 1, [506].log_data[15].valid := 1, [506].log_data[16].valid := 1, [506].log_data[17].valid := 1, [506].log_data[18].valid := 1, [506].log_data[19].valid := 1, [506].time.Year := 2023, [506].time.Month := 1, [506].time.Day := 11, [506].time.Hour := 10, [506].time.Minute := 34, [506].time.Second := 59, [507].log_data[0].min := 1.0, [507].log_data[0].max := 1.0, [507].log_data[0].total := 300.0, [507].log_data[0].time := 300.0, [507].log_data[0].minminute := 35, [507].log_data[0].maxminute := 35, [507].log_data[0].valid := 1, [507].log_data[1].valid := 1, [507].log_data[2].valid := 1, [507].log_data[3].valid := 1, [507].log_data[4].valid := 1, [507].log_data[5].valid := 1, [507].log_data[6].valid := 1, [507].log_data[7].valid := 1, [507].log_data[8].valid := 1, [507].log_data[9].valid := 1, [507].log_data[10].valid := 1, [507].log_data[11].valid := 1, [507].log_data[12].valid := 1, [507].log_data[13].valid := 1, [507].log_data[14].valid := 1, [507].log_data[15].valid := 1, [507].log_data[16].valid := 1, [507].log_data[17].valid := 1, [507].log_data[18].valid := 1, [507].log_data[19].valid := 1,
        [507].time.Year := 2023, [507].time.Month := 1, [507].time.Day := 11, [507].time.Hour := 10, [507].time.Minute := 39, [507].time.Second := 59, [508].log_data[0].min := 1.0, [508].log_data[0].max := 1.0, [508].log_data[0].total := 300.0, [508].log_data[0].time := 300.0, [508].log_data[0].minminute := 40, [508].log_data[0].maxminute := 40, [508].log_data[0].valid := 1, [508].log_data[1].valid := 1, [508].log_data[2].valid := 1, [508].log_data[3].valid := 1, [508].log_data[4].valid := 1, [508].log_data[5].valid := 1, [508].log_data[6].valid := 1, [508].log_data[7].valid := 1, [508].log_data[8].valid := 1, [508].log_data[9].valid := 1, [508].log_data[10].valid := 1, [508].log_data[11].valid := 1, [508].log_data[12].valid := 1, [508].log_data[13].valid := 1, [508].log_data[14].valid := 1, [508].log_data[15].valid := 1, [508].log_data[16].valid := 1, [508].log_data[17].valid := 1, [508].log_data[18].valid := 1, [508].log_data[19].valid := 1, [508].time.Year := 2023, [508].time.Month := 1, [508].time.Day := 11, [508].time.Hour := 10, [508].time.Minute := 44, [508].time.Second := 59, [509].log_data[0].min := 1.0, [509].log_data[0].max := 1.0, [509].log_data[0].total := 300.0, [509].log_data[0].time := 300.0, [509].log_data[0].minminute := 45, [509].log_data[0].maxminute := 45, [509].log_data[0].valid := 1, [509].log_data[1].valid := 1, [509].log_data[2].valid := 1, [509].log_data[3].valid := 1, [509].log_data[4].valid := 1, [509].log_data[5].valid := 1, [509].log_data[6].valid := 1, [509].log_data[7].valid := 1, [509].log_data[8].valid := 1, [509].log_data[9].valid := 1, [509].log_data[10].valid := 1, [509].log_data[11].valid := 1, [509].log_data[12].valid := 1, [509].log_data[13].valid := 1, [509].log_data[14].valid := 1, [509].log_data[15].valid := 1,
        [509].log_data[16].valid := 1, [509].log_data[17].valid := 1, [509].log_data[18].valid := 1, [509].log_data[19].valid := 1, [509].time.Year := 2023, [509].time.Month := 1, [509].time.Day := 11, [509].time.Hour := 10, [509].time.Minute := 49, [509].time.Second := 59, [510].log_data[0].min := 1.0, [510].log_data[0].max := 1.0, [510].log_data[0].total := 300.0, [510].log_data[0].time := 300.0, [510].log_data[0].minminute := 50, [510].log_data[0].maxminute := 50, [510].log_data[0].valid := 1, [510].log_data[1].valid := 1, [510].log_data[2].valid := 1, [510].log_data[3].valid := 1, [510].log_data[4].valid := 1, [510].log_data[5].valid := 1, [510].log_data[6].valid := 1, [510].log_data[7].valid := 1, [510].log_data[8].valid := 1, [510].log_data[9].valid := 1, [510].log_data[10].valid := 1, [510].log_data[11].valid := 1, [510].log_data[12].valid := 1, [510].log_data[13].valid := 1, [510].log_data[14].valid := 1, [510].log_data[15].valid := 1, [510].log_data[16].valid := 1, [510].log_data[17].valid := 1, [510].log_data[18].valid := 1, [510].log_data[19].valid := 1, [510].time.Year := 2023, [510].time.Month := 1, [510].time.Day := 11, [510].time.Hour := 10, [510].time.Minute := 54, [510].time.Second := 59, [511].log_data[0].min := 1.0, [511].log_data[0].max := 1.0, [511].log_data[0].total := 300.0, [511].log_data[0].time := 300.0, [511].log_data[0].minminute := 55, [511].log_data[0].maxminute := 55, [511].log_data[0].valid := 1, [511].log_data[1].valid := 1, [511].log_data[2].valid := 1, [511].log_data[3].valid := 1, [511].log_data[4].valid := 1, [511].log_data[5].valid := 1, [511].log_data[6].valid := 1, [511].log_data[7].valid := 1, [511].log_data[8].valid := 1, [511].log_data[9].valid := 1, [511].log_data[10].valid := 1, [511].log_data[11].valid := 1,
        [511].log_data[12].valid := 1, [511].log_data[13].valid := 1, [511].log_data[14].valid := 1, [511].log_data[15].valid := 1, [511].log_data[16].valid := 1, [511].log_data[17].valid := 1, [511].log_data[18].valid := 1, [511].log_data[19].valid := 1, [511].time.Year := 2023, [511].time.Month := 1, [511].time.Day := 11, [511].time.Hour := 10, [511].time.Minute := 59, [511].time.Second := 59, [512].log_data[0].min := 1.0, [512].log_data[0].max := 1.0, [512].log_data[0].total := 300.0, [512].log_data[0].time := 300.0, [512].log_data[0].valid := 1, [512].log_data[1].valid := 1, [512].log_data[2].valid := 1, [512].log_data[3].valid := 1, [512].log_data[4].valid := 1, [512].log_data[5].valid := 1, [512].log_data[6].valid := 1, [512].log_data[7].valid := 1, [512].log_data[8].valid := 1, [512].log_data[9].valid := 1, [512].log_data[10].valid := 1, [512].log_data[11].valid := 1, [512].log_data[12].valid := 1, [512].log_data[13].valid := 1, [512].log_data[14].valid := 1, [512].log_data[15].valid := 1, [512].log_data[16].valid := 1, [512].log_data[17].valid := 1, [512].log_data[18].valid := 1, [512].log_data[19].valid := 1, [512].time.Year := 2023, [512].time.Month := 1, [512].time.Day := 11, [512].time.Hour := 11, [512].time.Minute := 4, [512].time.Second := 59, [513].log_data[0].min := 1.0, [513].log_data[0].max := 1.0, [513].log_data[0].total := 300.0, [513].log_data[0].time := 300.0, [513].log_data[0].minminute := 5, [513].log_data[0].maxminute := 5, [513].log_data[0].valid := 1, [513].log_data[1].valid := 1, [513].log_data[2].valid := 1, [513].log_data[3].valid := 1, [513].log_data[4].valid := 1, [513].log_data[5].valid := 1, [513].log_data[6].valid := 1, [513].log_data[7].valid := 1, [513].log_data[8].valid := 1, [513].log_data[9].valid := 1,
        [513].log_data[10].valid := 1, [513].log_data[11].valid := 1, [513].log_data[12].valid := 1, [513].log_data[13].valid := 1, [513].log_data[14].valid := 1, [513].log_data[15].valid := 1, [513].log_data[16].valid := 1, [513].log_data[17].valid := 1, [513].log_data[18].valid := 1, [513].log_data[19].valid := 1, [513].time.Year := 2023, [513].time.Month := 1, [513].time.Day := 11, [513].time.Hour := 11, [513].time.Minute := 9, [513].time.Second := 59, [514].log_data[0].min := 1.0, [514].log_data[0].max := 1.0, [514].log_data[0].total := 300.0, [514].log_data[0].time := 300.0, [514].log_data[0].minminute := 10, [514].log_data[0].maxminute := 10, [514].log_data[0].valid := 1, [514].log_data[1].valid := 1, [514].log_data[2].valid := 1, [514].log_data[3].valid := 1, [514].log_data[4].valid := 1, [514].log_data[5].valid := 1, [514].log_data[6].valid := 1, [514].log_data[7].valid := 1, [514].log_data[8].valid := 1, [514].log_data[9].valid := 1, [514].log_data[10].valid := 1, [514].log_data[11].valid := 1, [514].log_data[12].valid := 1, [514].log_data[13].valid := 1, [514].log_data[14].valid := 1, [514].log_data[15].valid := 1, [514].log_data[16].valid := 1, [514].log_data[17].valid := 1, [514].log_data[18].valid := 1, [514].log_data[19].valid := 1, [514].time.Year := 2023, [514].time.Month := 1, [514].time.Day := 11, [514].time.Hour := 11, [514].time.Minute := 14, [514].time.Second := 59, [515].log_data[0].min := 1.0, [515].log_data[0].max := 1.0, [515].log_data[0].total := 300.0, [515].log_data[0].time := 300.0, [515].log_data[0].minminute := 15, [515].log_data[0].maxminute := 15, [515].log_data[0].valid := 1, [515].log_data[1].valid := 1, [515].log_data[2].valid := 1, [515].log_data[3].valid := 1, [515].log_data[4].valid := 1, [515].log_data[5].valid := 1,
        [515].log_data[6].valid := 1, [515].log_data[7].valid := 1, [515].log_data[8].valid := 1, [515].log_data[9].valid := 1, [515].log_data[10].valid := 1, [515].log_data[11].valid := 1, [515].log_data[12].valid := 1, [515].log_data[13].valid := 1, [515].log_data[14].valid := 1, [515].log_data[15].valid := 1, [515].log_data[16].valid := 1, [515].log_data[17].valid := 1, [515].log_data[18].valid := 1, [515].log_data[19].valid := 1, [515].time.Year := 2023, [515].time.Month := 1, [515].time.Day := 11, [515].time.Hour := 11, [515].time.Minute := 19, [515].time.Second := 59, [516].log_data[0].min := 1.0, [516].log_data[0].max := 1.0, [516].log_data[0].total := 300.0, [516].log_data[0].time := 300.0, [516].log_data[0].minminute := 20, [516].log_data[0].maxminute := 20, [516].log_data[0].valid := 1, [516].log_data[1].valid := 1, [516].log_data[2].valid := 1, [516].log_data[3].valid := 1, [516].log_data[4].valid := 1, [516].log_data[5].valid := 1, [516].log_data[6].valid := 1, [516].log_data[7].valid := 1, [516].log_data[8].valid := 1, [516].log_data[9].valid := 1, [516].log_data[10].valid := 1, [516].log_data[11].valid := 1, [516].log_data[12].valid := 1, [516].log_data[13].valid := 1, [516].log_data[14].valid := 1, [516].log_data[15].valid := 1, [516].log_data[16].valid := 1, [516].log_data[17].valid := 1, [516].log_data[18].valid := 1, [516].log_data[19].valid := 1, [516].time.Year := 2023, [516].time.Month := 1, [516].time.Day := 11, [516].time.Hour := 11, [516].time.Minute := 24, [516].time.Second := 59, [517].log_data[0].min := 1.0, [517].log_data[0].max := 1.0, [517].log_data[0].total := 300.0, [517].log_data[0].time := 300.0, [517].log_data[0].minminute := 25, [517].log_data[0].maxminute := 25, [517].log_data[0].valid := 1, [517].log_data[1].valid := 1,
        [517].log_data[2].valid := 1, [517].log_data[3].valid := 1, [517].log_data[4].valid := 1, [517].log_data[5].valid := 1, [517].log_data[6].valid := 1, [517].log_data[7].valid := 1, [517].log_data[8].valid := 1, [517].log_data[9].valid := 1, [517].log_data[10].valid := 1, [517].log_data[11].valid := 1, [517].log_data[12].valid := 1, [517].log_data[13].valid := 1, [517].log_data[14].valid := 1, [517].log_data[15].valid := 1, [517].log_data[16].valid := 1, [517].log_data[17].valid := 1, [517].log_data[18].valid := 1, [517].log_data[19].valid := 1, [517].time.Year := 2023, [517].time.Month := 1, [517].time.Day := 11, [517].time.Hour := 11, [517].time.Minute := 29, [517].time.Second := 59, [518].log_data[0].min := 1.0, [518].log_data[0].max := 1.0, [518].log_data[0].total := 300.0, [518].log_data[0].time := 300.0, [518].log_data[0].minminute := 30, [518].log_data[0].maxminute := 30, [518].log_data[0].valid := 1, [518].log_data[1].valid := 1, [518].log_data[2].valid := 1, [518].log_data[3].valid := 1, [518].log_data[4].valid := 1, [518].log_data[5].valid := 1, [518].log_data[6].valid := 1, [518].log_data[7].valid := 1, [518].log_data[8].valid := 1, [518].log_data[9].valid := 1, [518].log_data[10].valid := 1, [518].log_data[11].valid := 1, [518].log_data[12].valid := 1, [518].log_data[13].valid := 1, [518].log_data[14].valid := 1, [518].log_data[15].valid := 1, [518].log_data[16].valid := 1, [518].log_data[17].valid := 1, [518].log_data[18].valid := 1, [518].log_data[19].valid := 1, [518].time.Year := 2023, [518].time.Month := 1, [518].time.Day := 11, [518].time.Hour := 11, [518].time.Minute := 34, [518].time.Second := 59, [519].log_data[0].min := 1.0, [519].log_data[0].max := 1.0, [519].log_data[0].total := 300.0, [519].log_data[0].time := 300.0,
        [519].log_data[0].minminute := 35, [519].log_data[0].maxminute := 35, [519].log_data[0].valid := 1, [519].log_data[1].valid := 1, [519].log_data[2].valid := 1, [519].log_data[3].valid := 1, [519].log_data[4].valid := 1, [519].log_data[5].valid := 1, [519].log_data[6].valid := 1, [519].log_data[7].valid := 1, [519].log_data[8].valid := 1, [519].log_data[9].valid := 1, [519].log_data[10].valid := 1, [519].log_data[11].valid := 1, [519].log_data[12].valid := 1, [519].log_data[13].valid := 1, [519].log_data[14].valid := 1, [519].log_data[15].valid := 1, [519].log_data[16].valid := 1, [519].log_data[17].valid := 1, [519].log_data[18].valid := 1, [519].log_data[19].valid := 1, [519].time.Year := 2023, [519].time.Month := 1, [519].time.Day := 11, [519].time.Hour := 11, [519].time.Minute := 39, [519].time.Second := 59, [520].log_data[0].min := 1.0, [520].log_data[0].max := 1.0, [520].log_data[0].total := 300.0, [520].log_data[0].time := 300.0, [520].log_data[0].minminute := 40, [520].log_data[0].maxminute := 40, [520].log_data[0].valid := 1, [520].log_data[1].valid := 1, [520].log_data[2].valid := 1, [520].log_data[3].valid := 1, [520].log_data[4].valid := 1, [520].log_data[5].valid := 1, [520].log_data[6].valid := 1, [520].log_data[7].valid := 1, [520].log_data[8].valid := 1, [520].log_data[9].valid := 1, [520].log_data[10].valid := 1, [520].log_data[11].valid := 1, [520].log_data[12].valid := 1, [520].log_data[13].valid := 1, [520].log_data[14].valid := 1, [520].log_data[15].valid := 1, [520].log_data[16].valid := 1, [520].log_data[17].valid := 1, [520].log_data[18].valid := 1, [520].log_data[19].valid := 1, [520].time.Year := 2023, [520].time.Month := 1, [520].time.Day := 11, [520].time.Hour := 11, [520].time.Minute := 44, [520].time.Second := 59,
        [521].log_data[0].min := 1.0, [521].log_data[0].max := 1.0, [521].log_data[0].total := 300.0, [521].log_data[0].time := 300.0, [521].log_data[0].minminute := 45, [521].log_data[0].maxminute := 45, [521].log_data[0].valid := 1, [521].log_data[1].valid := 1, [521].log_data[2].valid := 1, [521].log_data[3].valid := 1, [521].log_data[4].valid := 1, [521].log_data[5].valid := 1, [521].log_data[6].valid := 1, [521].log_data[7].valid := 1, [521].log_data[8].valid := 1, [521].log_data[9].valid := 1, [521].log_data[10].valid := 1, [521].log_data[11].valid := 1, [521].log_data[12].valid := 1, [521].log_data[13].valid := 1, [521].log_data[14].valid := 1, [521].log_data[15].valid := 1, [521].log_data[16].valid := 1, [521].log_data[17].valid := 1, [521].log_data[18].valid := 1, [521].log_data[19].valid := 1, [521].time.Year := 2023, [521].time.Month := 1, [521].time.Day := 11, [521].time.Hour := 11, [521].time.Minute := 49, [521].time.Second := 59, [522].log_data[0].min := 1.0, [522].log_data[0].max := 1.0, [522].log_data[0].total := 300.0, [522].log_data[0].time := 300.0, [522].log_data[0].minminute := 50, [522].log_data[0].maxminute := 50, [522].log_data[0].valid := 1, [522].log_data[1].valid := 1, [522].log_data[2].valid := 1, [522].log_data[3].valid := 1, [522].log_data[4].valid := 1, [522].log_data[5].valid := 1, [522].log_data[6].valid := 1, [522].log_data[7].valid := 1, [522].log_data[8].valid := 1, [522].log_data[9].valid := 1, [522].log_data[10].valid := 1, [522].log_data[11].valid := 1, [522].log_data[12].valid := 1, [522].log_data[13].valid := 1, [522].log_data[14].valid := 1, [522].log_data[15].valid := 1, [522].log_data[16].valid := 1, [522].log_data[17].valid := 1, [522].log_data[18].valid := 1, [522].log_data[19].valid := 1, [522].time.Year := 2023, [522].time.Month := 1,
        [522].time.Day := 11, [522].time.Hour := 11, [522].time.Minute := 54, [522].time.Second := 59, [523].log_data[0].min := 1.0, [523].log_data[0].max := 1.0, [523].log_data[0].total := 300.0, [523].log_data[0].time := 300.0, [523].log_data[0].minminute := 55, [523].log_data[0].maxminute := 55, [523].log_data[0].valid := 1, [523].log_data[1].valid := 1, [523].log_data[2].valid := 1, [523].log_data[3].valid := 1, [523].log_data[4].valid := 1, [523].log_data[5].valid := 1, [523].log_data[6].valid := 1, [523].log_data[7].valid := 1, [523].log_data[8].valid := 1, [523].log_data[9].valid := 1, [523].log_data[10].valid := 1, [523].log_data[11].valid := 1, [523].log_data[12].valid := 1, [523].log_data[13].valid := 1, [523].log_data[14].valid := 1, [523].log_data[15].valid := 1, [523].log_data[16].valid := 1, [523].log_data[17].valid := 1, [523].log_data[18].valid := 1, [523].log_data[19].valid := 1, [523].time.Year := 2023, [523].time.Month := 1, [523].time.Day := 11, [523].time.Hour := 11, [523].time.Minute := 59, [523].time.Second := 59, [524].log_data[0].min := 1.0, [524].log_data[0].max := 1.0, [524].log_data[0].total := 300.0, [524].log_data[0].time := 300.0, [524].log_data[0].valid := 1, [524].log_data[1].valid := 1, [524].log_data[2].valid := 1, [524].log_data[3].valid := 1, [524].log_data[4].valid := 1, [524].log_data[5].valid := 1, [524].log_data[6].valid := 1, [524].log_data[7].valid := 1, [524].log_data[8].valid := 1, [524].log_data[9].valid := 1, [524].log_data[10].valid := 1, [524].log_data[11].valid := 1, [524].log_data[12].valid := 1, [524].log_data[13].valid := 1, [524].log_data[14].valid := 1, [524].log_data[15].valid := 1, [524].log_data[16].valid := 1, [524].log_data[17].valid := 1, [524].log_data[18].valid := 1, [524].log_data[19].valid := 1,
        [524].time.Year := 2023, [524].time.Month := 1, [524].time.Day := 11, [524].time.Hour := 12, [524].time.Minute := 4, [524].time.Second := 59, [525].log_data[0].min := 1.0, [525].log_data[0].max := 1.0, [525].log_data[0].total := 300.0, [525].log_data[0].time := 300.0, [525].log_data[0].minminute := 5, [525].log_data[0].maxminute := 5, [525].log_data[0].valid := 1, [525].log_data[1].valid := 1, [525].log_data[2].valid := 1, [525].log_data[3].valid := 1, [525].log_data[4].valid := 1, [525].log_data[5].valid := 1, [525].log_data[6].valid := 1, [525].log_data[7].valid := 1, [525].log_data[8].valid := 1, [525].log_data[9].valid := 1, [525].log_data[10].valid := 1, [525].log_data[11].valid := 1, [525].log_data[12].valid := 1, [525].log_data[13].valid := 1, [525].log_data[14].valid := 1, [525].log_data[15].valid := 1, [525].log_data[16].valid := 1, [525].log_data[17].valid := 1, [525].log_data[18].valid := 1, [525].log_data[19].valid := 1, [525].time.Year := 2023, [525].time.Month := 1, [525].time.Day := 11, [525].time.Hour := 12, [525].time.Minute := 9, [525].time.Second := 59, [526].log_data[0].min := 1.0, [526].log_data[0].max := 1.0, [526].log_data[0].total := 300.0, [526].log_data[0].time := 300.0, [526].log_data[0].minminute := 10, [526].log_data[0].maxminute := 10, [526].log_data[0].valid := 1, [526].log_data[1].valid := 1, [526].log_data[2].valid := 1, [526].log_data[3].valid := 1, [526].log_data[4].valid := 1, [526].log_data[5].valid := 1, [526].log_data[6].valid := 1, [526].log_data[7].valid := 1, [526].log_data[8].valid := 1, [526].log_data[9].valid := 1, [526].log_data[10].valid := 1, [526].log_data[11].valid := 1, [526].log_data[12].valid := 1, [526].log_data[13].valid := 1, [526].log_data[14].valid := 1, [526].log_data[15].valid := 1,
        [526].log_data[16].valid := 1, [526].log_data[17].valid := 1, [526].log_data[18].valid := 1, [526].log_data[19].valid := 1, [526].time.Year := 2023, [526].time.Month := 1, [526].time.Day := 11, [526].time.Hour := 12, [526].time.Minute := 14, [526].time.Second := 59, [527].log_data[0].min := 1.0, [527].log_data[0].max := 1.0, [527].log_data[0].total := 300.0, [527].log_data[0].time := 300.0, [527].log_data[0].minminute := 15, [527].log_data[0].maxminute := 15, [527].log_data[0].valid := 1, [527].log_data[1].valid := 1, [527].log_data[2].valid := 1, [527].log_data[3].valid := 1, [527].log_data[4].valid := 1, [527].log_data[5].valid := 1, [527].log_data[6].valid := 1, [527].log_data[7].valid := 1, [527].log_data[8].valid := 1, [527].log_data[9].valid := 1, [527].log_data[10].valid := 1, [527].log_data[11].valid := 1, [527].log_data[12].valid := 1, [527].log_data[13].valid := 1, [527].log_data[14].valid := 1, [527].log_data[15].valid := 1, [527].log_data[16].valid := 1, [527].log_data[17].valid := 1, [527].log_data[18].valid := 1, [527].log_data[19].valid := 1, [527].time.Year := 2023, [527].time.Month := 1, [527].time.Day := 11, [527].time.Hour := 12, [527].time.Minute := 19, [527].time.Second := 59, [528].log_data[0].min := 1.0, [528].log_data[0].max := 1.0, [528].log_data[0].total := 300.0, [528].log_data[0].time := 300.0, [528].log_data[0].minminute := 20, [528].log_data[0].maxminute := 20, [528].log_data[0].valid := 1, [528].log_data[1].valid := 1, [528].log_data[2].valid := 1, [528].log_data[3].valid := 1, [528].log_data[4].valid := 1, [528].log_data[5].valid := 1, [528].log_data[6].valid := 1, [528].log_data[7].valid := 1, [528].log_data[8].valid := 1, [528].log_data[9].valid := 1, [528].log_data[10].valid := 1, [528].log_data[11].valid := 1,
        [528].log_data[12].valid := 1, [528].log_data[13].valid := 1, [528].log_data[14].valid := 1, [528].log_data[15].valid := 1, [528].log_data[16].valid := 1, [528].log_data[17].valid := 1, [528].log_data[18].valid := 1, [528].log_data[19].valid := 1, [528].time.Year := 2023, [528].time.Month := 1, [528].time.Day := 11, [528].time.Hour := 12, [528].time.Minute := 24, [528].time.Second := 59, [529].log_data[0].min := 1.0, [529].log_data[0].max := 1.0, [529].log_data[0].total := 300.0, [529].log_data[0].time := 300.0, [529].log_data[0].minminute := 25, [529].log_data[0].maxminute := 25, [529].log_data[0].valid := 1, [529].log_data[1].valid := 1, [529].log_data[2].valid := 1, [529].log_data[3].valid := 1, [529].log_data[4].valid := 1, [529].log_data[5].valid := 1, [529].log_data[6].valid := 1, [529].log_data[7].valid := 1, [529].log_data[8].valid := 1, [529].log_data[9].valid := 1, [529].log_data[10].valid := 1, [529].log_data[11].valid := 1, [529].log_data[12].valid := 1, [529].log_data[13].valid := 1, [529].log_data[14].valid := 1, [529].log_data[15].valid := 1, [529].log_data[16].valid := 1, [529].log_data[17].valid := 1, [529].log_data[18].valid := 1, [529].log_data[19].valid := 1, [529].time.Year := 2023, [529].time.Month := 1, [529].time.Day := 11, [529].time.Hour := 12, [529].time.Minute := 29, [529].time.Second := 59, [530].log_data[0].min := 1.0, [530].log_data[0].max := 1.0, [530].log_data[0].total := 300.0, [530].log_data[0].time := 300.0, [530].log_data[0].minminute := 30, [530].log_data[0].maxminute := 30, [530].log_data[0].valid := 1, [530].log_data[1].valid := 1, [530].log_data[2].valid := 1, [530].log_data[3].valid := 1, [530].log_data[4].valid := 1, [530].log_data[5].valid := 1, [530].log_data[6].valid := 1, [530].log_data[7].valid := 1,
        [530].log_data[8].valid := 1, [530].log_data[9].valid := 1, [530].log_data[10].valid := 1, [530].log_data[11].valid := 1, [530].log_data[12].valid := 1, [530].log_data[13].valid := 1, [530].log_data[14].valid := 1, [530].log_data[15].valid := 1, [530].log_data[16].valid := 1, [530].log_data[17].valid := 1, [530].log_data[18].valid := 1, [530].log_data[19].valid := 1, [530].time.Year := 2023, [530].time.Month := 1, [530].time.Day := 11, [530].time.Hour := 12, [530].time.Minute := 34, [530].time.Second := 59, [531].log_data[0].min := 1.0, [531].log_data[0].max := 1.0, [531].log_data[0].total := 300.0, [531].log_data[0].time := 300.0, [531].log_data[0].minminute := 35, [531].log_data[0].maxminute := 35, [531].log_data[0].valid := 1, [531].log_data[1].valid := 1, [531].log_data[2].valid := 1, [531].log_data[3].valid := 1, [531].log_data[4].valid := 1, [531].log_data[5].valid := 1, [531].log_data[6].valid := 1, [531].log_data[7].valid := 1, [531].log_data[8].valid := 1, [531].log_data[9].valid := 1, [531].log_data[10].valid := 1, [531].log_data[11].valid := 1, [531].log_data[12].valid := 1, [531].log_data[13].valid := 1, [531].log_data[14].valid := 1, [531].log_data[15].valid := 1, [531].log_data[16].valid := 1, [531].log_data[17].valid := 1, [531].log_data[18].valid := 1, [531].log_data[19].valid := 1, [531].time.Year := 2023, [531].time.Month := 1, [531].time.Day := 11, [531].time.Hour := 12, [531].time.Minute := 39, [531].time.Second := 59, [532].log_data[0].min := 1.0, [532].log_data[0].max := 1.0, [532].log_data[0].total := 300.0, [532].log_data[0].time := 300.0, [532].log_data[0].minminute := 40, [532].log_data[0].maxminute := 40, [532].log_data[0].valid := 1, [532].log_data[1].valid := 1, [532].log_data[2].valid := 1, [532].log_data[3].valid := 1,
        [532].log_data[4].valid := 1, [532].log_data[5].valid := 1, [532].log_data[6].valid := 1, [532].log_data[7].valid := 1, [532].log_data[8].valid := 1, [532].log_data[9].valid := 1, [532].log_data[10].valid := 1, [532].log_data[11].valid := 1, [532].log_data[12].valid := 1, [532].log_data[13].valid := 1, [532].log_data[14].valid := 1, [532].log_data[15].valid := 1, [532].log_data[16].valid := 1, [532].log_data[17].valid := 1, [532].log_data[18].valid := 1, [532].log_data[19].valid := 1, [532].time.Year := 2023, [532].time.Month := 1, [532].time.Day := 11, [532].time.Hour := 12, [532].time.Minute := 44, [532].time.Second := 59, [533].log_data[0].min := 1.0, [533].log_data[0].max := 1.0, [533].log_data[0].total := 300.0, [533].log_data[0].time := 300.0, [533].log_data[0].minminute := 45, [533].log_data[0].maxminute := 45, [533].log_data[0].valid := 1, [533].log_data[1].valid := 1, [533].log_data[2].valid := 1, [533].log_data[3].valid := 1, [533].log_data[4].valid := 1, [533].log_data[5].valid := 1, [533].log_data[6].valid := 1, [533].log_data[7].valid := 1, [533].log_data[8].valid := 1, [533].log_data[9].valid := 1, [533].log_data[10].valid := 1, [533].log_data[11].valid := 1, [533].log_data[12].valid := 1, [533].log_data[13].valid := 1, [533].log_data[14].valid := 1, [533].log_data[15].valid := 1, [533].log_data[16].valid := 1, [533].log_data[17].valid := 1, [533].log_data[18].valid := 1, [533].log_data[19].valid := 1, [533].time.Year := 2023, [533].time.Month := 1, [533].time.Day := 11, [533].time.Hour := 12, [533].time.Minute := 49, [533].time.Second := 59, [534].log_data[0].min := 1.0, [534].log_data[0].max := 1.0, [534].log_data[0].total := 300.0, [534].log_data[0].time := 300.0, [534].log_data[0].minminute := 50, [534].log_data[0].maxminute := 50,
        [534].log_data[0].valid := 1, [534].log_data[1].valid := 1, [534].log_data[2].valid := 1, [534].log_data[3].valid := 1, [534].log_data[4].valid := 1, [534].log_data[5].valid := 1, [534].log_data[6].valid := 1, [534].log_data[7].valid := 1, [534].log_data[8].valid := 1, [534].log_data[9].valid := 1, [534].log_data[10].valid := 1, [534].log_data[11].valid := 1, [534].log_data[12].valid := 1, [534].log_data[13].valid := 1, [534].log_data[14].valid := 1, [534].log_data[15].valid := 1, [534].log_data[16].valid := 1, [534].log_data[17].valid := 1, [534].log_data[18].valid := 1, [534].log_data[19].valid := 1, [534].time.Year := 2023, [534].time.Month := 1, [534].time.Day := 11, [534].time.Hour := 12, [534].time.Minute := 54, [534].time.Second := 59, [535].log_data[0].min := 1.0, [535].log_data[0].max := 1.0, [535].log_data[0].total := 300.0, [535].log_data[0].time := 300.0, [535].log_data[0].minminute := 55, [535].log_data[0].maxminute := 55, [535].log_data[0].valid := 1, [535].log_data[1].valid := 1, [535].log_data[2].valid := 1, [535].log_data[3].valid := 1, [535].log_data[4].valid := 1, [535].log_data[5].valid := 1, [535].log_data[6].valid := 1, [535].log_data[7].valid := 1, [535].log_data[8].valid := 1, [535].log_data[9].valid := 1, [535].log_data[10].valid := 1, [535].log_data[11].valid := 1, [535].log_data[12].valid := 1, [535].log_data[13].valid := 1, [535].log_data[14].valid := 1, [535].log_data[15].valid := 1, [535].log_data[16].valid := 1, [535].log_data[17].valid := 1, [535].log_data[18].valid := 1, [535].log_data[19].valid := 1, [535].time.Year := 2023, [535].time.Month := 1, [535].time.Day := 11, [535].time.Hour := 12, [535].time.Minute := 59, [535].time.Second := 59, [536].log_data[0].min := 1.0, [536].log_data[0].max := 1.0,
        [536].log_data[0].total := 300.0, [536].log_data[0].time := 300.0, [536].log_data[0].valid := 1, [536].log_data[1].valid := 1, [536].log_data[2].valid := 1, [536].log_data[3].valid := 1, [536].log_data[4].valid := 1, [536].log_data[5].valid := 1, [536].log_data[6].valid := 1, [536].log_data[7].valid := 1, [536].log_data[8].valid := 1, [536].log_data[9].valid := 1, [536].log_data[10].valid := 1, [536].log_data[11].valid := 1, [536].log_data[12].valid := 1, [536].log_data[13].valid := 1, [536].log_data[14].valid := 1, [536].log_data[15].valid := 1, [536].log_data[16].valid := 1, [536].log_data[17].valid := 1, [536].log_data[18].valid := 1, [536].log_data[19].valid := 1, [536].time.Year := 2023, [536].time.Month := 1, [536].time.Day := 11, [536].time.Hour := 13, [536].time.Minute := 4, [536].time.Second := 59, [537].log_data[0].min := 1.0, [537].log_data[0].max := 1.0, [537].log_data[0].total := 300.0, [537].log_data[0].time := 300.0, [537].log_data[0].minminute := 5, [537].log_data[0].maxminute := 5, [537].log_data[0].valid := 1, [537].log_data[1].valid := 1, [537].log_data[2].valid := 1, [537].log_data[3].valid := 1, [537].log_data[4].valid := 1, [537].log_data[5].valid := 1, [537].log_data[6].valid := 1, [537].log_data[7].valid := 1, [537].log_data[8].valid := 1, [537].log_data[9].valid := 1, [537].log_data[10].valid := 1, [537].log_data[11].valid := 1, [537].log_data[12].valid := 1, [537].log_data[13].valid := 1, [537].log_data[14].valid := 1, [537].log_data[15].valid := 1, [537].log_data[16].valid := 1, [537].log_data[17].valid := 1, [537].log_data[18].valid := 1, [537].log_data[19].valid := 1, [537].time.Year := 2023, [537].time.Month := 1, [537].time.Day := 11, [537].time.Hour := 13, [537].time.Minute := 9, [537].time.Second := 59,
        [538].log_data[0].min := 1.0, [538].log_data[0].max := 1.0, [538].log_data[0].total := 300.0, [538].log_data[0].time := 300.0, [538].log_data[0].minminute := 10, [538].log_data[0].maxminute := 10, [538].log_data[0].valid := 1, [538].log_data[1].valid := 1, [538].log_data[2].valid := 1, [538].log_data[3].valid := 1, [538].log_data[4].valid := 1, [538].log_data[5].valid := 1, [538].log_data[6].valid := 1, [538].log_data[7].valid := 1, [538].log_data[8].valid := 1, [538].log_data[9].valid := 1, [538].log_data[10].valid := 1, [538].log_data[11].valid := 1, [538].log_data[12].valid := 1, [538].log_data[13].valid := 1, [538].log_data[14].valid := 1, [538].log_data[15].valid := 1, [538].log_data[16].valid := 1, [538].log_data[17].valid := 1, [538].log_data[18].valid := 1, [538].log_data[19].valid := 1, [538].time.Year := 2023, [538].time.Month := 1, [538].time.Day := 11, [538].time.Hour := 13, [538].time.Minute := 14, [538].time.Second := 59, [539].log_data[0].min := 1.0, [539].log_data[0].max := 1.0, [539].log_data[0].total := 300.0, [539].log_data[0].time := 300.0, [539].log_data[0].minminute := 15, [539].log_data[0].maxminute := 15, [539].log_data[0].valid := 1, [539].log_data[1].valid := 1, [539].log_data[2].valid := 1, [539].log_data[3].valid := 1, [539].log_data[4].valid := 1, [539].log_data[5].valid := 1, [539].log_data[6].valid := 1, [539].log_data[7].valid := 1, [539].log_data[8].valid := 1, [539].log_data[9].valid := 1, [539].log_data[10].valid := 1, [539].log_data[11].valid := 1, [539].log_data[12].valid := 1, [539].log_data[13].valid := 1, [539].log_data[14].valid := 1, [539].log_data[15].valid := 1, [539].log_data[16].valid := 1, [539].log_data[17].valid := 1, [539].log_data[18].valid := 1, [539].log_data[19].valid := 1, [539].time.Year := 2023, [539].time.Month := 1,
        [539].time.Day := 11, [539].time.Hour := 13, [539].time.Minute := 19, [539].time.Second := 59, [540].log_data[0].min := 1.0, [540].log_data[0].max := 1.0, [540].log_data[0].total := 300.0, [540].log_data[0].time := 300.0, [540].log_data[0].minminute := 20, [540].log_data[0].maxminute := 20, [540].log_data[0].valid := 1, [540].log_data[1].valid := 1, [540].log_data[2].valid := 1, [540].log_data[3].valid := 1, [540].log_data[4].valid := 1, [540].log_data[5].valid := 1, [540].log_data[6].valid := 1, [540].log_data[7].valid := 1, [540].log_data[8].valid := 1, [540].log_data[9].valid := 1, [540].log_data[10].valid := 1, [540].log_data[11].valid := 1, [540].log_data[12].valid := 1, [540].log_data[13].valid := 1, [540].log_data[14].valid := 1, [540].log_data[15].valid := 1, [540].log_data[16].valid := 1, [540].log_data[17].valid := 1, [540].log_data[18].valid := 1, [540].log_data[19].valid := 1, [540].time.Year := 2023, [540].time.Month := 1, [540].time.Day := 11, [540].time.Hour := 13, [540].time.Minute := 24, [540].time.Second := 59, [541].log_data[0].min := 1.0, [541].log_data[0].max := 1.0, [541].log_data[0].total := 300.0, [541].log_data[0].time := 300.0, [541].log_data[0].minminute := 25, [541].log_data[0].maxminute := 25, [541].log_data[0].valid := 1, [541].log_data[1].valid := 1, [541].log_data[2].valid := 1, [541].log_data[3].valid := 1, [541].log_data[4].valid := 1, [541].log_data[5].valid := 1, [541].log_data[6].valid := 1, [541].log_data[7].valid := 1, [541].log_data[8].valid := 1, [541].log_data[9].valid := 1, [541].log_data[10].valid := 1, [541].log_data[11].valid := 1, [541].log_data[12].valid := 1, [541].log_data[13].valid := 1, [541].log_data[14].valid := 1, [541].log_data[15].valid := 1, [541].log_data[16].valid := 1, [541].log_data[17].valid := 1,
        [541].log_data[18].valid := 1, [541].log_data[19].valid := 1, [541].time.Year := 2023, [541].time.Month := 1, [541].time.Day := 11, [541].time.Hour := 13, [541].time.Minute := 29, [541].time.Second := 59, [542].log_data[0].min := 1.0, [542].log_data[0].max := 1.0, [542].log_data[0].total := 300.0, [542].log_data[0].time := 300.0, [542].log_data[0].minminute := 30, [542].log_data[0].maxminute := 30, [542].log_data[0].valid := 1, [542].log_data[1].valid := 1, [542].log_data[2].valid := 1, [542].log_data[3].valid := 1, [542].log_data[4].valid := 1, [542].log_data[5].valid := 1, [542].log_data[6].valid := 1, [542].log_data[7].valid := 1, [542].log_data[8].valid := 1, [542].log_data[9].valid := 1, [542].log_data[10].valid := 1, [542].log_data[11].valid := 1, [542].log_data[12].valid := 1, [542].log_data[13].valid := 1, [542].log_data[14].valid := 1, [542].log_data[15].valid := 1, [542].log_data[16].valid := 1, [542].log_data[17].valid := 1, [542].log_data[18].valid := 1, [542].log_data[19].valid := 1, [542].time.Year := 2023, [542].time.Month := 1, [542].time.Day := 11, [542].time.Hour := 13, [542].time.Minute := 34, [542].time.Second := 59, [543].log_data[0].min := 1.0, [543].log_data[0].max := 1.0, [543].log_data[0].total := 300.0, [543].log_data[0].time := 300.0, [543].log_data[0].minminute := 35, [543].log_data[0].maxminute := 35, [543].log_data[0].valid := 1, [543].log_data[1].valid := 1, [543].log_data[2].valid := 1, [543].log_data[3].valid := 1, [543].log_data[4].valid := 1, [543].log_data[5].valid := 1, [543].log_data[6].valid := 1, [543].log_data[7].valid := 1, [543].log_data[8].valid := 1, [543].log_data[9].valid := 1, [543].log_data[10].valid := 1, [543].log_data[11].valid := 1, [543].log_data[12].valid := 1, [543].log_data[13].valid := 1,
        [543].log_data[14].valid := 1, [543].log_data[15].valid := 1, [543].log_data[16].valid := 1, [543].log_data[17].valid := 1, [543].log_data[18].valid := 1, [543].log_data[19].valid := 1, [543].time.Year := 2023, [543].time.Month := 1, [543].time.Day := 11, [543].time.Hour := 13, [543].time.Minute := 39, [543].time.Second := 59, [544].log_data[0].min := 1.0, [544].log_data[0].max := 1.0, [544].log_data[0].total := 300.0, [544].log_data[0].time := 300.0, [544].log_data[0].minminute := 40, [544].log_data[0].maxminute := 40, [544].log_data[0].valid := 1, [544].log_data[1].valid := 1, [544].log_data[2].valid := 1, [544].log_data[3].valid := 1, [544].log_data[4].valid := 1, [544].log_data[5].valid := 1, [544].log_data[6].valid := 1, [544].log_data[7].valid := 1, [544].log_data[8].valid := 1, [544].log_data[9].valid := 1, [544].log_data[10].valid := 1, [544].log_data[11].valid := 1, [544].log_data[12].valid := 1, [544].log_data[13].valid := 1, [544].log_data[14].valid := 1, [544].log_data[15].valid := 1, [544].log_data[16].valid := 1, [544].log_data[17].valid := 1, [544].log_data[18].valid := 1, [544].log_data[19].valid := 1, [544].time.Year := 2023, [544].time.Month := 1, [544].time.Day := 11, [544].time.Hour := 13, [544].time.Minute := 44, [544].time.Second := 59, [545].log_data[0].min := 1.0, [545].log_data[0].max := 1.0, [545].log_data[0].total := 300.0, [545].log_data[0].time := 300.0, [545].log_data[0].minminute := 45, [545].log_data[0].maxminute := 45, [545].log_data[0].valid := 1, [545].log_data[1].valid := 1, [545].log_data[2].valid := 1, [545].log_data[3].valid := 1, [545].log_data[4].valid := 1, [545].log_data[5].valid := 1, [545].log_data[6].valid := 1, [545].log_data[7].valid := 1, [545].log_data[8].valid := 1, [545].log_data[9].valid := 1,
        [545].log_data[10].valid := 1, [545].log_data[11].valid := 1, [545].log_data[12].valid := 1, [545].log_data[13].valid := 1, [545].log_data[14].valid := 1, [545].log_data[15].valid := 1, [545].log_data[16].valid := 1, [545].log_data[17].valid := 1, [545].log_data[18].valid := 1, [545].log_data[19].valid := 1, [545].time.Year := 2023, [545].time.Month := 1, [545].time.Day := 11, [545].time.Hour := 13, [545].time.Minute := 49, [545].time.Second := 59, [546].log_data[0].min := 1.0, [546].log_data[0].max := 1.0, [546].log_data[0].total := 300.0, [546].log_data[0].time := 300.0, [546].log_data[0].minminute := 50, [546].log_data[0].maxminute := 50, [546].log_data[0].valid := 1, [546].log_data[1].valid := 1, [546].log_data[2].valid := 1, [546].log_data[3].valid := 1, [546].log_data[4].valid := 1, [546].log_data[5].valid := 1, [546].log_data[6].valid := 1, [546].log_data[7].valid := 1, [546].log_data[8].valid := 1, [546].log_data[9].valid := 1, [546].log_data[10].valid := 1, [546].log_data[11].valid := 1, [546].log_data[12].valid := 1, [546].log_data[13].valid := 1, [546].log_data[14].valid := 1, [546].log_data[15].valid := 1, [546].log_data[16].valid := 1, [546].log_data[17].valid := 1, [546].log_data[18].valid := 1, [546].log_data[19].valid := 1, [546].time.Year := 2023, [546].time.Month := 1, [546].time.Day := 11, [546].time.Hour := 13, [546].time.Minute := 54, [546].time.Second := 59, [547].log_data[0].min := 1.0, [547].log_data[0].max := 1.0, [547].log_data[0].total := 300.0, [547].log_data[0].time := 300.0, [547].log_data[0].minminute := 55, [547].log_data[0].maxminute := 55, [547].log_data[0].valid := 1, [547].log_data[1].valid := 1, [547].log_data[2].valid := 1, [547].log_data[3].valid := 1, [547].log_data[4].valid := 1, [547].log_data[5].valid := 1,
        [547].log_data[6].valid := 1, [547].log_data[7].valid := 1, [547].log_data[8].valid := 1, [547].log_data[9].valid := 1, [547].log_data[10].valid := 1, [547].log_data[11].valid := 1, [547].log_data[12].valid := 1, [547].log_data[13].valid := 1, [547].log_data[14].valid := 1, [547].log_data[15].valid := 1, [547].log_data[16].valid := 1, [547].log_data[17].valid := 1, [547].log_data[18].valid := 1, [547].log_data[19].valid := 1, [547].time.Year := 2023, [547].time.Month := 1, [547].time.Day := 11, [547].time.Hour := 13, [547].time.Minute := 59, [547].time.Second := 59, [548].log_data[0].min := 1.0, [548].log_data[0].max := 1.0, [548].log_data[0].total := 299.5, [548].log_data[0].time := 299.5, [548].log_data[0].valid := 1, [548].log_data[1].valid := 1, [548].log_data[2].valid := 1, [548].log_data[3].valid := 1, [548].log_data[4].valid := 1, [548].log_data[5].valid := 1, [548].log_data[6].valid := 1, [548].log_data[7].valid := 1, [548].log_data[8].valid := 1, [548].log_data[9].valid := 1, [548].log_data[10].valid := 1, [548].log_data[11].valid := 1, [548].log_data[12].valid := 1, [548].log_data[13].valid := 1, [548].log_data[14].valid := 1, [548].log_data[15].valid := 1, [548].log_data[16].valid := 1, [548].log_data[17].valid := 1, [548].log_data[18].valid := 1, [548].log_data[19].valid := 1, [548].time.Year := 2023, [548].time.Month := 1, [548].time.Day := 11, [548].time.Hour := 14, [548].time.Minute := 4, [548].time.Second := 59, [549].log_data[0].min := 1.0, [549].log_data[0].max := 1.0, [549].log_data[0].total := 300.0, [549].log_data[0].time := 300.0, [549].log_data[0].minminute := 5, [549].log_data[0].maxminute := 5, [549].log_data[0].valid := 1, [549].log_data[1].valid := 1, [549].log_data[2].valid := 1, [549].log_data[3].valid := 1,
        [549].log_data[4].valid := 1, [549].log_data[5].valid := 1, [549].log_data[6].valid := 1, [549].log_data[7].valid := 1, [549].log_data[8].valid := 1, [549].log_data[9].valid := 1, [549].log_data[10].valid := 1, [549].log_data[11].valid := 1, [549].log_data[12].valid := 1, [549].log_data[13].valid := 1, [549].log_data[14].valid := 1, [549].log_data[15].valid := 1, [549].log_data[16].valid := 1, [549].log_data[17].valid := 1, [549].log_data[18].valid := 1, [549].log_data[19].valid := 1, [549].time.Year := 2023, [549].time.Month := 1, [549].time.Day := 11, [549].time.Hour := 14, [549].time.Minute := 9, [549].time.Second := 59, [550].log_data[0].min := 1.0, [550].log_data[0].max := 1.0, [550].log_data[0].total := 300.0, [550].log_data[0].time := 300.0, [550].log_data[0].minminute := 10, [550].log_data[0].maxminute := 10, [550].log_data[0].valid := 1, [550].log_data[1].valid := 1, [550].log_data[2].valid := 1, [550].log_data[3].valid := 1, [550].log_data[4].valid := 1, [550].log_data[5].valid := 1, [550].log_data[6].valid := 1, [550].log_data[7].valid := 1, [550].log_data[8].valid := 1, [550].log_data[9].valid := 1, [550].log_data[10].valid := 1, [550].log_data[11].valid := 1, [550].log_data[12].valid := 1, [550].log_data[13].valid := 1, [550].log_data[14].valid := 1, [550].log_data[15].valid := 1, [550].log_data[16].valid := 1, [550].log_data[17].valid := 1, [550].log_data[18].valid := 1, [550].log_data[19].valid := 1, [550].time.Year := 2023, [550].time.Month := 1, [550].time.Day := 11, [550].time.Hour := 14, [550].time.Minute := 14, [550].time.Second := 59, [551].log_data[0].min := 1.0, [551].log_data[0].max := 1.0, [551].log_data[0].total := 300.0, [551].log_data[0].time := 300.0, [551].log_data[0].minminute := 15, [551].log_data[0].maxminute := 15,
        [551].log_data[0].valid := 1, [551].log_data[1].valid := 1, [551].log_data[2].valid := 1, [551].log_data[3].valid := 1, [551].log_data[4].valid := 1, [551].log_data[5].valid := 1, [551].log_data[6].valid := 1, [551].log_data[7].valid := 1, [551].log_data[8].valid := 1, [551].log_data[9].valid := 1, [551].log_data[10].valid := 1, [551].log_data[11].valid := 1, [551].log_data[12].valid := 1, [551].log_data[13].valid := 1, [551].log_data[14].valid := 1, [551].log_data[15].valid := 1, [551].log_data[16].valid := 1, [551].log_data[17].valid := 1, [551].log_data[18].valid := 1, [551].log_data[19].valid := 1, [551].time.Year := 2023, [551].time.Month := 1, [551].time.Day := 11, [551].time.Hour := 14, [551].time.Minute := 19, [551].time.Second := 59, [552].log_data[0].min := 1.0, [552].log_data[0].max := 1.0, [552].log_data[0].total := 300.0, [552].log_data[0].time := 300.0, [552].log_data[0].minminute := 20, [552].log_data[0].maxminute := 20, [552].log_data[0].valid := 1, [552].log_data[1].valid := 1, [552].log_data[2].valid := 1, [552].log_data[3].valid := 1, [552].log_data[4].valid := 1, [552].log_data[5].valid := 1, [552].log_data[6].valid := 1, [552].log_data[7].valid := 1, [552].log_data[8].valid := 1, [552].log_data[9].valid := 1, [552].log_data[10].valid := 1, [552].log_data[11].valid := 1, [552].log_data[12].valid := 1, [552].log_data[13].valid := 1, [552].log_data[14].valid := 1, [552].log_data[15].valid := 1, [552].log_data[16].valid := 1, [552].log_data[17].valid := 1, [552].log_data[18].valid := 1, [552].log_data[19].valid := 1, [552].time.Year := 2023, [552].time.Month := 1, [552].time.Day := 11, [552].time.Hour := 14, [552].time.Minute := 24, [552].time.Second := 59, [553].log_data[0].min := 1.0, [553].log_data[0].max := 1.0,
        [553].log_data[0].total := 300.0, [553].log_data[0].time := 300.0, [553].log_data[0].minminute := 25, [553].log_data[0].maxminute := 25, [553].log_data[0].valid := 1, [553].log_data[1].valid := 1, [553].log_data[2].valid := 1, [553].log_data[3].valid := 1, [553].log_data[4].valid := 1, [553].log_data[5].valid := 1, [553].log_data[6].valid := 1, [553].log_data[7].valid := 1, [553].log_data[8].valid := 1, [553].log_data[9].valid := 1, [553].log_data[10].valid := 1, [553].log_data[11].valid := 1, [553].log_data[12].valid := 1, [553].log_data[13].valid := 1, [553].log_data[14].valid := 1, [553].log_data[15].valid := 1, [553].log_data[16].valid := 1, [553].log_data[17].valid := 1, [553].log_data[18].valid := 1, [553].log_data[19].valid := 1, [553].time.Year := 2023, [553].time.Month := 1, [553].time.Day := 11, [553].time.Hour := 14, [553].time.Minute := 29, [553].time.Second := 59, [554].log_data[0].min := 1.0, [554].log_data[0].max := 1.0, [554].log_data[0].total := 300.0, [554].log_data[0].time := 300.0, [554].log_data[0].minminute := 30, [554].log_data[0].maxminute := 30, [554].log_data[0].valid := 1, [554].log_data[1].valid := 1, [554].log_data[2].valid := 1, [554].log_data[3].valid := 1, [554].log_data[4].valid := 1, [554].log_data[5].valid := 1, [554].log_data[6].valid := 1, [554].log_data[7].valid := 1, [554].log_data[8].valid := 1, [554].log_data[9].valid := 1, [554].log_data[10].valid := 1, [554].log_data[11].valid := 1, [554].log_data[12].valid := 1, [554].log_data[13].valid := 1, [554].log_data[14].valid := 1, [554].log_data[15].valid := 1, [554].log_data[16].valid := 1, [554].log_data[17].valid := 1, [554].log_data[18].valid := 1, [554].log_data[19].valid := 1, [554].time.Year := 2023, [554].time.Month := 1, [554].time.Day := 11, [554].time.Hour := 14,
        [554].time.Minute := 34, [554].time.Second := 59, [555].log_data[0].min := 1.0, [555].log_data[0].max := 1.0, [555].log_data[0].total := 300.0, [555].log_data[0].time := 300.0, [555].log_data[0].minminute := 35, [555].log_data[0].maxminute := 35, [555].log_data[0].valid := 1, [555].log_data[1].valid := 1, [555].log_data[2].valid := 1, [555].log_data[3].valid := 1, [555].log_data[4].valid := 1, [555].log_data[5].valid := 1, [555].log_data[6].valid := 1, [555].log_data[7].valid := 1, [555].log_data[8].valid := 1, [555].log_data[9].valid := 1, [555].log_data[10].valid := 1, [555].log_data[11].valid := 1, [555].log_data[12].valid := 1, [555].log_data[13].valid := 1, [555].log_data[14].valid := 1, [555].log_data[15].valid := 1, [555].log_data[16].valid := 1, [555].log_data[17].valid := 1, [555].log_data[18].valid := 1, [555].log_data[19].valid := 1, [555].time.Year := 2023, [555].time.Month := 1, [555].time.Day := 11, [555].time.Hour := 14, [555].time.Minute := 39, [555].time.Second := 59, [556].log_data[0].min := 1.0, [556].log_data[0].max := 1.0, [556].log_data[0].total := 300.0, [556].log_data[0].time := 300.0, [556].log_data[0].minminute := 40, [556].log_data[0].maxminute := 40, [556].log_data[0].valid := 1, [556].log_data[1].valid := 1, [556].log_data[2].valid := 1, [556].log_data[3].valid := 1, [556].log_data[4].valid := 1, [556].log_data[5].valid := 1, [556].log_data[6].valid := 1, [556].log_data[7].valid := 1, [556].log_data[8].valid := 1, [556].log_data[9].valid := 1, [556].log_data[10].valid := 1, [556].log_data[11].valid := 1, [556].log_data[12].valid := 1, [556].log_data[13].valid := 1, [556].log_data[14].valid := 1, [556].log_data[15].valid := 1, [556].log_data[16].valid := 1, [556].log_data[17].valid := 1, [556].log_data[18].valid := 1, [556].log_data[19].valid := 1,
        [556].time.Year := 2023, [556].time.Month := 1, [556].time.Day := 11, [556].time.Hour := 14, [556].time.Minute := 44, [556].time.Second := 59, [557].log_data[0].min := 1.0, [557].log_data[0].max := 1.0, [557].log_data[0].total := 300.0, [557].log_data[0].time := 300.0, [557].log_data[0].minminute := 45, [557].log_data[0].maxminute := 45, [557].log_data[0].valid := 1, [557].log_data[1].valid := 1, [557].log_data[2].valid := 1, [557].log_data[3].valid := 1, [557].log_data[4].valid := 1, [557].log_data[5].valid := 1, [557].log_data[6].valid := 1, [557].log_data[7].valid := 1, [557].log_data[8].valid := 1, [557].log_data[9].valid := 1, [557].log_data[10].valid := 1, [557].log_data[11].valid := 1, [557].log_data[12].valid := 1, [557].log_data[13].valid := 1, [557].log_data[14].valid := 1, [557].log_data[15].valid := 1, [557].log_data[16].valid := 1, [557].log_data[17].valid := 1, [557].log_data[18].valid := 1, [557].log_data[19].valid := 1, [557].time.Year := 2023, [557].time.Month := 1, [557].time.Day := 11, [557].time.Hour := 14, [557].time.Minute := 49, [557].time.Second := 59, [558].log_data[0].min := 1.0, [558].log_data[0].max := 1.0, [558].log_data[0].total := 300.0, [558].log_data[0].time := 300.0, [558].log_data[0].minminute := 50, [558].log_data[0].maxminute := 50, [558].log_data[0].valid := 1, [558].log_data[1].valid := 1, [558].log_data[2].valid := 1, [558].log_data[3].valid := 1, [558].log_data[4].valid := 1, [558].log_data[5].valid := 1, [558].log_data[6].valid := 1, [558].log_data[7].valid := 1, [558].log_data[8].valid := 1, [558].log_data[9].valid := 1, [558].log_data[10].valid := 1, [558].log_data[11].valid := 1, [558].log_data[12].valid := 1, [558].log_data[13].valid := 1, [558].log_data[14].valid := 1, [558].log_data[15].valid := 1,
        [558].log_data[16].valid := 1, [558].log_data[17].valid := 1, [558].log_data[18].valid := 1, [558].log_data[19].valid := 1, [558].time.Year := 2023, [558].time.Month := 1, [558].time.Day := 11, [558].time.Hour := 14, [558].time.Minute := 54, [558].time.Second := 59, [559].log_data[0].min := 1.0, [559].log_data[0].max := 1.0, [559].log_data[0].total := 300.0, [559].log_data[0].time := 300.0, [559].log_data[0].minminute := 55, [559].log_data[0].maxminute := 55, [559].log_data[0].valid := 1, [559].log_data[1].valid := 1, [559].log_data[2].valid := 1, [559].log_data[3].valid := 1, [559].log_data[4].valid := 1, [559].log_data[5].valid := 1, [559].log_data[6].valid := 1, [559].log_data[7].valid := 1, [559].log_data[8].valid := 1, [559].log_data[9].valid := 1, [559].log_data[10].valid := 1, [559].log_data[11].valid := 1, [559].log_data[12].valid := 1, [559].log_data[13].valid := 1, [559].log_data[14].valid := 1, [559].log_data[15].valid := 1, [559].log_data[16].valid := 1, [559].log_data[17].valid := 1, [559].log_data[18].valid := 1, [559].log_data[19].valid := 1, [559].time.Year := 2023, [559].time.Month := 1, [559].time.Day := 11, [559].time.Hour := 14, [559].time.Minute := 59, [559].time.Second := 59, [560].log_data[0].min := 1.0, [560].log_data[0].max := 1.0, [560].log_data[0].total := 300.0, [560].log_data[0].time := 300.0, [560].log_data[0].valid := 1, [560].log_data[1].valid := 1, [560].log_data[2].valid := 1, [560].log_data[3].valid := 1, [560].log_data[4].valid := 1, [560].log_data[5].valid := 1, [560].log_data[6].valid := 1, [560].log_data[7].valid := 1, [560].log_data[8].valid := 1, [560].log_data[9].valid := 1, [560].log_data[10].valid := 1, [560].log_data[11].valid := 1, [560].log_data[12].valid := 1, [560].log_data[13].valid := 1,
        [560].log_data[14].valid := 1, [560].log_data[15].valid := 1, [560].log_data[16].valid := 1, [560].log_data[17].valid := 1, [560].log_data[18].valid := 1, [560].log_data[19].valid := 1, [560].time.Year := 2023, [560].time.Month := 1, [560].time.Day := 11, [560].time.Hour := 15, [560].time.Minute := 4, [560].time.Second := 59, [561].log_data[0].min := 1.0, [561].log_data[0].max := 1.0, [561].log_data[0].total := 300.0, [561].log_data[0].time := 300.0, [561].log_data[0].minminute := 5, [561].log_data[0].maxminute := 5, [561].log_data[0].valid := 1, [561].log_data[1].valid := 1, [561].log_data[2].valid := 1, [561].log_data[3].valid := 1, [561].log_data[4].valid := 1, [561].log_data[5].valid := 1, [561].log_data[6].valid := 1, [561].log_data[7].valid := 1, [561].log_data[8].valid := 1, [561].log_data[9].valid := 1, [561].log_data[10].valid := 1, [561].log_data[11].valid := 1, [561].log_data[12].valid := 1, [561].log_data[13].valid := 1, [561].log_data[14].valid := 1, [561].log_data[15].valid := 1, [561].log_data[16].valid := 1, [561].log_data[17].valid := 1, [561].log_data[18].valid := 1, [561].log_data[19].valid := 1, [561].time.Year := 2023, [561].time.Month := 1, [561].time.Day := 11, [561].time.Hour := 15, [561].time.Minute := 9, [561].time.Second := 59, [562].log_data[0].min := 1.0, [562].log_data[0].max := 1.0, [562].log_data[0].total := 300.0, [562].log_data[0].time := 300.0, [562].log_data[0].minminute := 10, [562].log_data[0].maxminute := 10, [562].log_data[0].valid := 1, [562].log_data[1].valid := 1, [562].log_data[2].valid := 1, [562].log_data[3].valid := 1, [562].log_data[4].valid := 1, [562].log_data[5].valid := 1, [562].log_data[6].valid := 1, [562].log_data[7].valid := 1, [562].log_data[8].valid := 1, [562].log_data[9].valid := 1,
        [562].log_data[10].valid := 1, [562].log_data[11].valid := 1, [562].log_data[12].valid := 1, [562].log_data[13].valid := 1, [562].log_data[14].valid := 1, [562].log_data[15].valid := 1, [562].log_data[16].valid := 1, [562].log_data[17].valid := 1, [562].log_data[18].valid := 1, [562].log_data[19].valid := 1, [562].time.Year := 2023, [562].time.Month := 1, [562].time.Day := 11, [562].time.Hour := 15, [562].time.Minute := 14, [562].time.Second := 59, [563].log_data[0].min := 1.0, [563].log_data[0].max := 1.0, [563].log_data[0].total := 300.0, [563].log_data[0].time := 300.0, [563].log_data[0].minminute := 15, [563].log_data[0].maxminute := 15, [563].log_data[0].valid := 1, [563].log_data[1].valid := 1, [563].log_data[2].valid := 1, [563].log_data[3].valid := 1, [563].log_data[4].valid := 1, [563].log_data[5].valid := 1, [563].log_data[6].valid := 1, [563].log_data[7].valid := 1, [563].log_data[8].valid := 1, [563].log_data[9].valid := 1, [563].log_data[10].valid := 1, [563].log_data[11].valid := 1, [563].log_data[12].valid := 1, [563].log_data[13].valid := 1, [563].log_data[14].valid := 1, [563].log_data[15].valid := 1, [563].log_data[16].valid := 1, [563].log_data[17].valid := 1, [563].log_data[18].valid := 1, [563].log_data[19].valid := 1, [563].time.Year := 2023, [563].time.Month := 1, [563].time.Day := 11, [563].time.Hour := 15, [563].time.Minute := 19, [563].time.Second := 59, [564].log_data[0].min := 1.0, [564].log_data[0].max := 1.0, [564].log_data[0].total := 300.0, [564].log_data[0].time := 300.0, [564].log_data[0].minminute := 20, [564].log_data[0].maxminute := 20, [564].log_data[0].valid := 1, [564].log_data[1].valid := 1, [564].log_data[2].valid := 1, [564].log_data[3].valid := 1, [564].log_data[4].valid := 1, [564].log_data[5].valid := 1,
        [564].log_data[6].valid := 1, [564].log_data[7].valid := 1, [564].log_data[8].valid := 1, [564].log_data[9].valid := 1, [564].log_data[10].valid := 1, [564].log_data[11].valid := 1, [564].log_data[12].valid := 1, [564].log_data[13].valid := 1, [564].log_data[14].valid := 1, [564].log_data[15].valid := 1, [564].log_data[16].valid := 1, [564].log_data[17].valid := 1, [564].log_data[18].valid := 1, [564].log_data[19].valid := 1, [564].time.Year := 2023, [564].time.Month := 1, [564].time.Day := 11, [564].time.Hour := 15, [564].time.Minute := 24, [564].time.Second := 59, [565].log_data[0].min := 1.0, [565].log_data[0].max := 1.0, [565].log_data[0].total := 300.0, [565].log_data[0].time := 300.0, [565].log_data[0].minminute := 25, [565].log_data[0].maxminute := 25, [565].log_data[0].valid := 1, [565].log_data[1].valid := 1, [565].log_data[2].valid := 1, [565].log_data[3].valid := 1, [565].log_data[4].valid := 1, [565].log_data[5].valid := 1, [565].log_data[6].valid := 1, [565].log_data[7].valid := 1, [565].log_data[8].valid := 1, [565].log_data[9].valid := 1, [565].log_data[10].valid := 1, [565].log_data[11].valid := 1, [565].log_data[12].valid := 1, [565].log_data[13].valid := 1, [565].log_data[14].valid := 1, [565].log_data[15].valid := 1, [565].log_data[16].valid := 1, [565].log_data[17].valid := 1, [565].log_data[18].valid := 1, [565].log_data[19].valid := 1, [565].time.Year := 2023, [565].time.Month := 1, [565].time.Day := 11, [565].time.Hour := 15, [565].time.Minute := 29, [565].time.Second := 59, [566].log_data[0].min := 1.0, [566].log_data[0].max := 1.0, [566].log_data[0].total := 300.0, [566].log_data[0].time := 300.0, [566].log_data[0].minminute := 30, [566].log_data[0].maxminute := 30, [566].log_data[0].valid := 1, [566].log_data[1].valid := 1,
        [566].log_data[2].valid := 1, [566].log_data[3].valid := 1, [566].log_data[4].valid := 1, [566].log_data[5].valid := 1, [566].log_data[6].valid := 1, [566].log_data[7].valid := 1, [566].log_data[8].valid := 1, [566].log_data[9].valid := 1, [566].log_data[10].valid := 1, [566].log_data[11].valid := 1, [566].log_data[12].valid := 1, [566].log_data[13].valid := 1, [566].log_data[14].valid := 1, [566].log_data[15].valid := 1, [566].log_data[16].valid := 1, [566].log_data[17].valid := 1, [566].log_data[18].valid := 1, [566].log_data[19].valid := 1, [566].time.Year := 2023, [566].time.Month := 1, [566].time.Day := 11, [566].time.Hour := 15, [566].time.Minute := 34, [566].time.Second := 59, [567].log_data[0].min := 1.0, [567].log_data[0].max := 1.0, [567].log_data[0].total := 300.0, [567].log_data[0].time := 300.0, [567].log_data[0].minminute := 35, [567].log_data[0].maxminute := 35, [567].log_data[0].valid := 1, [567].log_data[1].valid := 1, [567].log_data[2].valid := 1, [567].log_data[3].valid := 1, [567].log_data[4].valid := 1, [567].log_data[5].valid := 1, [567].log_data[6].valid := 1, [567].log_data[7].valid := 1, [567].log_data[8].valid := 1, [567].log_data[9].valid := 1, [567].log_data[10].valid := 1, [567].log_data[11].valid := 1, [567].log_data[12].valid := 1, [567].log_data[13].valid := 1, [567].log_data[14].valid := 1, [567].log_data[15].valid := 1, [567].log_data[16].valid := 1, [567].log_data[17].valid := 1, [567].log_data[18].valid := 1, [567].log_data[19].valid := 1, [567].time.Year := 2023, [567].time.Month := 1, [567].time.Day := 11, [567].time.Hour := 15, [567].time.Minute := 39, [567].time.Second := 59, [568].log_data[0].min := 1.0, [568].log_data[0].max := 1.0, [568].log_data[0].total := 300.0, [568].log_data[0].time := 300.0,
        [568].log_data[0].minminute := 40, [568].log_data[0].maxminute := 40, [568].log_data[0].valid := 1, [568].log_data[1].valid := 1, [568].log_data[2].valid := 1, [568].log_data[3].valid := 1, [568].log_data[4].valid := 1, [568].log_data[5].valid := 1, [568].log_data[6].valid := 1, [568].log_data[7].valid := 1, [568].log_data[8].valid := 1, [568].log_data[9].valid := 1, [568].log_data[10].valid := 1, [568].log_data[11].valid := 1, [568].log_data[12].valid := 1, [568].log_data[13].valid := 1, [568].log_data[14].valid := 1, [568].log_data[15].valid := 1, [568].log_data[16].valid := 1, [568].log_data[17].valid := 1, [568].log_data[18].valid := 1, [568].log_data[19].valid := 1, [568].time.Year := 2023, [568].time.Month := 1, [568].time.Day := 11, [568].time.Hour := 15, [568].time.Minute := 44, [568].time.Second := 59, [569].log_data[0].min := 1.0, [569].log_data[0].max := 1.0, [569].log_data[0].total := 300.0, [569].log_data[0].time := 300.0, [569].log_data[0].minminute := 45, [569].log_data[0].maxminute := 45, [569].log_data[0].valid := 1, [569].log_data[1].valid := 1, [569].log_data[2].valid := 1, [569].log_data[3].valid := 1, [569].log_data[4].valid := 1, [569].log_data[5].valid := 1, [569].log_data[6].valid := 1, [569].log_data[7].valid := 1, [569].log_data[8].valid := 1, [569].log_data[9].valid := 1, [569].log_data[10].valid := 1, [569].log_data[11].valid := 1, [569].log_data[12].valid := 1, [569].log_data[13].valid := 1, [569].log_data[14].valid := 1, [569].log_data[15].valid := 1, [569].log_data[16].valid := 1, [569].log_data[17].valid := 1, [569].log_data[18].valid := 1, [569].log_data[19].valid := 1, [569].time.Year := 2023, [569].time.Month := 1, [569].time.Day := 11, [569].time.Hour := 15, [569].time.Minute := 49, [569].time.Second := 59,
        [570].log_data[0].min := 1.0, [570].log_data[0].max := 1.0, [570].log_data[0].total := 300.0, [570].log_data[0].time := 300.0, [570].log_data[0].minminute := 50, [570].log_data[0].maxminute := 50, [570].log_data[0].valid := 1, [570].log_data[1].valid := 1, [570].log_data[2].valid := 1, [570].log_data[3].valid := 1, [570].log_data[4].valid := 1, [570].log_data[5].valid := 1, [570].log_data[6].valid := 1, [570].log_data[7].valid := 1, [570].log_data[8].valid := 1, [570].log_data[9].valid := 1, [570].log_data[10].valid := 1, [570].log_data[11].valid := 1, [570].log_data[12].valid := 1, [570].log_data[13].valid := 1, [570].log_data[14].valid := 1, [570].log_data[15].valid := 1, [570].log_data[16].valid := 1, [570].log_data[17].valid := 1, [570].log_data[18].valid := 1, [570].log_data[19].valid := 1, [570].time.Year := 2023, [570].time.Month := 1, [570].time.Day := 11, [570].time.Hour := 15, [570].time.Minute := 54, [570].time.Second := 59, [571].log_data[0].min := 1.0, [571].log_data[0].max := 1.0, [571].log_data[0].total := 300.0, [571].log_data[0].time := 300.0, [571].log_data[0].minminute := 55, [571].log_data[0].maxminute := 55, [571].log_data[0].valid := 1, [571].log_data[1].valid := 1, [571].log_data[2].valid := 1, [571].log_data[3].valid := 1, [571].log_data[4].valid := 1, [571].log_data[5].valid := 1, [571].log_data[6].valid := 1, [571].log_data[7].valid := 1, [571].log_data[8].valid := 1, [571].log_data[9].valid := 1, [571].log_data[10].valid := 1, [571].log_data[11].valid := 1, [571].log_data[12].valid := 1, [571].log_data[13].valid := 1, [571].log_data[14].valid := 1, [571].log_data[15].valid := 1, [571].log_data[16].valid := 1, [571].log_data[17].valid := 1, [571].log_data[18].valid := 1, [571].log_data[19].valid := 1, [571].time.Year := 2023, [571].time.Month := 1,
